LIN {X 0,Y 420.308,Z 548.759,A -85,B 0,C 180,E1 -10290.385,E2 -10290.385} C_VEL
LIN {X 0,Y 420.15,Z 551.033,A -85,B 0,C 180,E1 -10290.92,E2 -10290.92} C_VEL
LIN {X 0,Y 424.128,Z 570.244,A -85,B 0,C 180,E1 -10291.48,E2 -10291.48} C_VEL
LIN {X 0,Y 422.913,Z 658.502,A -85,B 0,C 180,E1 -10293.08,E2 -10293.08} C_VEL
LIN {X 0,Y 422.511,Z 671.225,A -85,B 0,C 180,E1 -10293.497,E2 -10293.497} C_VEL
LIN {X 0,Y 421.973,Z 684.045,A -85,B 0,C 180,E1 -10294.115,E2 -10294.115} C_VEL
LIN {X 0,Y 421.324,Z 696.249,A -85,B 0,C 180,E1 -10294.924,E2 -10294.924} C_VEL
LIN {X 0,Y 420.519,Z 708.11,A -85,B 0,C 180,E1 -10295.936,E2 -10295.936} C_VEL
LIN {X 0,Y 419.769,Z 718.542,A -85,B 0,C 180,E1 -10297.065,E2 -10297.065} C_VEL
LIN {X 0,Y 419.109,Z 728.059,A -85,B 0,C 180,E1 -10298.348,E2 -10298.348} C_VEL
LIN {X 0,Y 418.513,Z 735.947,A -85,B 0,C 180,E1 -10299.651,E2 -10299.651} C_VEL
LIN {X 0,Y 418,Z 742.497,A -85,B 0,C 180,E1 -10300.974,E2 -10300.974} C_VEL
LIN {X 0,Y 417.596,Z 749.006,A -85,B 0,C 180,E1 -10302.629,E2 -10302.629} C_VEL
LIN {X 0,Y 417.299,Z 754.023,A -85,B 0,C 180,E1 -10304.318,E2 -10304.318} C_VEL
LIN {X 0,Y 417.103,Z 757.009,A -85,B 0,C 180,E1 -10305.67,E2 -10305.67} C_VEL
LIN {X 0,Y 416.912,Z 759.823,A -85,B 0,C 180,E1 -10307.603,E2 -10307.603} C_VEL
LIN {X 0,Y 416.814,Z 760.935,A -85,B 0,C 180,E1 -10309.354,E2 -10309.354} C_VEL
LIN {X 0,Y 416.814,Z 760.853,A -85,B 0,C 180,E1 -10310.86,E2 -10310.86} C_VEL
LIN {X 0,Y 416.909,Z 759.474,A -85,B 0,C 180,E1 -10312.639,E2 -10312.639} C_VEL
LIN {X 0,Y 417.117,Z 756.524,A -85,B 0,C 180,E1 -10314.528,E2 -10314.528} C_VEL
LIN {X 0,Y 417.313,Z 752.371,A -85,B 0,C 180,E1 -10316.239,E2 -10316.239} C_VEL
LIN {X 0,Y 417.678,Z 746.51,A -85,B 0,C 180,E1 -10317.994,E2 -10317.994} C_VEL
LIN {X 0,Y 418.041,Z 740.528,A -85,B 0,C 180,E1 -10319.39,E2 -10319.39} C_VEL
LIN {X 0,Y 418.614,Z 732.644,A -85,B 0,C 180,E1 -10320.867,E2 -10320.867} C_VEL
LIN {X 0,Y 419.189,Z 723.962,A -85,B 0,C 180,E1 -10322.175,E2 -10322.175} C_VEL
LIN {X 0,Y 419.91,Z 713.909,A -85,B 0,C 180,E1 -10323.405,E2 -10323.405} C_VEL
LIN {X 0,Y 420.672,Z 703.331,A -85,B 0,C 180,E1 -10324.442,E2 -10324.442} C_VEL
LIN {X 0,Y 421.29,Z 691.58,A -85,B 0,C 180,E1 -10325.353,E2 -10325.353} C_VEL
LIN {X 0,Y 421.916,Z 679.248,A -85,B 0,C 180,E1 -10326.085,E2 -10326.085} C_VEL
LIN {X 0,Y 422.378,Z 666.034,A -85,B 0,C 180,E1 -10326.643,E2 -10326.643} C_VEL
LIN {X 0,Y 422.72,Z 652.404,A -85,B 0,C 180,E1 -10327.003,E2 -10327.003} C_VEL
LIN {X 0,Y 423.711,Z 575.673,A -85,B 0,C 180,E1 -10328.355,E2 -10328.355} C_VEL
LIN {X 0,Y 422.921,Z 571.915,A -85,B 0,C 180,E1 -10328.458,E2 -10328.458} C_VEL
LIN {X 0,Y 420.296,Z 567.48,A -85,B 0,C 180,E1 -10328.654,E2 -10328.654} C_VEL
LIN {X 0,Y 415.703,Z 561.063,A -85,B 0,C 180,E1 -10328.977,E2 -10328.977} C_VEL
LIN {X 0,Y 414.319,Z 557.368,A -85,B 0,C 180,E1 -10329.109,E2 -10329.109} C_VEL
LIN {X 0,Y 412.948,Z 550.435,A -85,B 0,C 180,E1 -10329.328,E2 -10329.328} C_VEL
LIN {X 0,Y 413.198,Z 543.912,A -85,B 0,C 180,E1 -10330.889,E2 -10330.889} C_VEL
LIN {X 0,Y 411.297,Z 533.254,A -85,B 0,C 180,E1 -10333.625,E2 -10333.625} C_VEL
LIN {X 0,Y 411.298,Z 533.253,A -85,B 0,C 180,E1 -10337.167,E2 -10337.167} C_VEL
LIN {X 0,Y 411.289,Z 533.25,A -85,B 0,C 180,E1 -10340.163,E2 -10340.163} C_VEL
LIN {X 0,Y 411.447,Z 533.233,A -85,B 0,C 180,E1 -10343.134,E2 -10343.134} C_VEL
LIN {X 0,Y 411.307,Z 533.251,A -85,B 0,C 180,E1 -10345.1,E2 -10345.1} C_VEL
LIN {X 0,Y 411.511,Z 533.221,A -85,B 0,C 180,E1 -10348.044,E2 -10348.044} C_VEL
LIN {X 0,Y 411.639,Z 533.205,A -85,B 0,C 180,E1 -10350.001,E2 -10350.001} C_VEL
LIN {X 0,Y 411.463,Z 533.235,A -85,B 0,C 180,E1 -10352.939,E2 -10352.939} C_VEL
LIN {X 0,Y 411.449,Z 533.235,A -85,B 0,C 180,E1 -10356.868,E2 -10356.868} C_VEL
LIN {X 0,Y 411.291,Z 533.248,A -85,B 0,C 180,E1 -10359.84,E2 -10359.84} C_VEL
LIN {X 0,Y 411.304,Z 533.254,A -85,B 0,C 180,E1 -10363.106,E2 -10363.106} C_VEL
LIN {X 0,Y 411.262,Z 533.257,A -85,B 0,C 180,E1 -10366.87,E2 -10366.87} C_VEL
LIN {X 0,Y 411.23,Z 533.256,A -85,B 0,C 180,E1 -10369.988,E2 -10369.988} C_VEL
LIN {X 0,Y 411.203,Z 533.267,A -85,B 0,C 180,E1 -10373.149,E2 -10373.149} C_VEL
LIN {X 0,Y 411.238,Z 533.255,A -85,B 0,C 180,E1 -10376.382,E2 -10376.382} C_VEL
LIN {X 0,Y 411.201,Z 533.261,A -85,B 0,C 180,E1 -10379.714,E2 -10379.714} C_VEL
LIN {X 0,Y 411.208,Z 533.265,A -85,B 0,C 180,E1 -10383.157,E2 -10383.157} C_VEL
LIN {X 0,Y 411.194,Z 533.261,A -85,B 0,C 180,E1 -10386.554,E2 -10386.554} C_VEL
LIN {X 0,Y 411.217,Z 533.26,A -85,B 0,C 180,E1 -10389.729,E2 -10389.729} C_VEL
LIN {X 0,Y 411.18,Z 533.267,A -85,B 0,C 180,E1 -10393.134,E2 -10393.134} C_VEL
LIN {X 0,Y 411.171,Z 533.265,A -85,B 0,C 180,E1 -10395.882,E2 -10395.882} C_VEL
LIN {X 0,Y 411.166,Z 533.265,A -85,B 0,C 180,E1 -10398.773,E2 -10398.773} C_VEL
LIN {X 0,Y 411.208,Z 533.262,A -85,B 0,C 180,E1 -10401.833,E2 -10401.833} C_VEL
LIN {X 0,Y 411.215,Z 533.261,A -85,B 0,C 180,E1 -10405.123,E2 -10405.123} C_VEL
LIN {X 0,Y 411.17,Z 533.265,A -85,B 0,C 180,E1 -10408.004,E2 -10408.004} C_VEL
LIN {X 0,Y 411.223,Z 533.263,A -85,B 0,C 180,E1 -10411.411,E2 -10411.411} C_VEL
LIN {X 0,Y 411.242,Z 533.261,A -85,B 0,C 180,E1 -10413.62,E2 -10413.62} C_VEL
LIN {X 0,Y 411.202,Z 533.26,A -85,B 0,C 180,E1 -10416.853,E2 -10416.853} C_VEL
LIN {X 0,Y 411.22,Z 533.26,A -85,B 0,C 180,E1 -10420.051,E2 -10420.051} C_VEL
LIN {X 0,Y 411.269,Z 533.253,A -85,B 0,C 180,E1 -10423.132,E2 -10423.132} C_VEL
LIN {X 0,Y 411.312,Z 533.246,A -85,B 0,C 180,E1 -10426.897,E2 -10426.897} C_VEL
LIN {X 0,Y 411.298,Z 533.25,A -85,B 0,C 180,E1 -10430.162,E2 -10430.162} C_VEL
LIN {X 0,Y 411.459,Z 533.228,A -85,B 0,C 180,E1 -10433.134,E2 -10433.134} C_VEL
LIN {X 0,Y 411.315,Z 533.246,A -85,B 0,C 180,E1 -10435.1,E2 -10435.1} C_VEL
LIN {X 0,Y 411.518,Z 533.225,A -85,B 0,C 180,E1 -10438.043,E2 -10438.043} C_VEL
LIN {X 0,Y 411.647,Z 533.209,A -85,B 0,C 180,E1 -10440.001,E2 -10440.001} C_VEL
LIN {X 0,Y 411.464,Z 533.227,A -85,B 0,C 180,E1 -10442.938,E2 -10442.938} C_VEL
LIN {X 0,Y 411.468,Z 533.226,A -85,B 0,C 180,E1 -10446.867,E2 -10446.867} C_VEL
LIN {X 0,Y 411.362,Z 533.24,A -85,B 0,C 180,E1 -10448.846,E2 -10448.846} C_VEL
LIN {X 0,Y 411.291,Z 533.255,A -85,B 0,C 180,E1 -10451.833,E2 -10451.833} C_VEL
LIN {X 0,Y 411.268,Z 533.251,A -85,B 0,C 180,E1 -10454.853,E2 -10454.853} C_VEL
LIN {X 0,Y 411.258,Z 533.259,A -85,B 0,C 180,E1 -10457.915,E2 -10457.915} C_VEL
LIN {X 0,Y 411.204,Z 533.259,A -85,B 0,C 180,E1 -10461.034,E2 -10461.034} C_VEL
LIN {X 0,Y 411.228,Z 533.262,A -85,B 0,C 180,E1 -10464.216,E2 -10464.216} C_VEL
LIN {X 0,Y 411.267,Z 533.252,A -85,B 0,C 180,E1 -10467.478,E2 -10467.478} C_VEL
LIN {X 0,Y 411.197,Z 533.261,A -85,B 0,C 180,E1 -10470.847,E2 -10470.847} C_VEL
LIN {X 0,Y 411.214,Z 533.263,A -85,B 0,C 180,E1 -10474.333,E2 -10474.333} C_VEL
LIN {X 0,Y 411.198,Z 533.264,A -85,B 0,C 180,E1 -10477.974,E2 -10477.974} C_VEL
LIN {X 0,Y 411.167,Z 533.264,A -85,B 0,C 180,E1 -10481.227,E2 -10481.227} C_VEL
LIN {X 0,Y 411.183,Z 533.267,A -85,B 0,C 180,E1 -10484.49,E2 -10484.49} C_VEL
LIN {X 0,Y 411.185,Z 533.268,A -85,B 0,C 180,E1 -10488.194,E2 -10488.194} C_VEL
LIN {X 0,Y 411.231,Z 533.258,A -85,B 0,C 180,E1 -10490.776,E2 -10490.776} C_VEL
LIN {X 0,Y 411.205,Z 533.266,A -85,B 0,C 180,E1 -10494.471,E2 -10494.471} C_VEL
LIN {X 0,Y 411.215,Z 533.26,A -85,B 0,C 180,E1 -10496.873,E2 -10496.873} C_VEL
LIN {X 0,Y 411.24,Z 533.261,A -85,B 0,C 180,E1 -10500.643,E2 -10500.643} C_VEL
LIN {X 0,Y 411.32,Z 533.412,A -85,B 0,C 180,E1 -10502.353,E2 -10502.353} C_VEL
LIN {X 0,Y 413.758,Z 545.682,A -85,B 0,C 180,E1 -10505.139,E2 -10505.139} C_VEL
LIN {X 0,Y 414.314,Z 549.496,A -85,B 0,C 180,E1 -10505.975,E2 -10505.975} C_VEL
LIN {X 0,Y 413.43,Z 563.343,A -85,B 0,C 180,E1 -10508.823,E2 -10508.823} C_VEL
LIN {X 0,Y 412.789,Z 572.615,A -85,B 0,C 180,E1 -10510.705,E2 -10510.705} C_VEL
LIN {X 0,Y 416.803,Z 598.62,A -85,B 0,C 180,E1 -10511.379,E2 -10511.379} C_VEL
LIN {X 0,Y 415.714,Z 681.281,A -85,B 0,C 180,E1 -10512.885,E2 -10512.885} C_VEL
LIN {X 0,Y 415.188,Z 695.012,A -85,B 0,C 180,E1 -10513.338,E2 -10513.338} C_VEL
LIN {X 0,Y 414.584,Z 707.414,A -85,B 0,C 180,E1 -10513.946,E2 -10513.946} C_VEL
LIN {X 0,Y 413.866,Z 719.311,A -85,B 0,C 180,E1 -10514.738,E2 -10514.738} C_VEL
LIN {X 0,Y 413.089,Z 730.763,A -85,B 0,C 180,E1 -10515.717,E2 -10515.717} C_VEL
LIN {X 0,Y 412.34,Z 741.085,A -85,B 0,C 180,E1 -10516.821,E2 -10516.821} C_VEL
LIN {X 0,Y 411.762,Z 749.532,A -85,B 0,C 180,E1 -10517.93,E2 -10517.93} C_VEL
LIN {X 0,Y 411.046,Z 758.685,A -85,B 0,C 180,E1 -10519.407,E2 -10519.407} C_VEL
LIN {X 0,Y 410.59,Z 766.062,A -85,B 0,C 180,E1 -10520.889,E2 -10520.889} C_VEL
LIN {X 0,Y 410.313,Z 771.055,A -85,B 0,C 180,E1 -10522.123,E2 -10522.123} C_VEL
LIN {X 0,Y 410.101,Z 776.187,A -85,B 0,C 180,E1 -10523.702,E2 -10523.702} C_VEL
LIN {X 0,Y 410.026,Z 779.603,A -85,B 0,C 180,E1 -10525.082,E2 -10525.082} C_VEL
LIN {X 0,Y 409.936,Z 781.513,A -85,B 0,C 180,E1 -10526.066,E2 -10526.066} C_VEL
LIN {X 0,Y 409.929,Z 782.966,A -85,B 0,C 180,E1 -10527.05,E2 -10527.05} C_VEL
LIN {X 0,Y 409.967,Z 783.99,A -85,B 0,C 180,E1 -10528.034,E2 -10528.034} C_VEL
LIN {X 0,Y 409.936,Z 784.617,A -85,B 0,C 180,E1 -10529.016,E2 -10529.016} C_VEL
LIN {X 0,Y 409.926,Z 784.853,A -85,B 0,C 180,E1 -10529.999,E2 -10529.999} C_VEL
LIN {X 0,Y 409.936,Z 784.659,A -85,B 0,C 180,E1 -10530.981,E2 -10530.981} C_VEL
LIN {X 0,Y 409.967,Z 784.052,A -85,B 0,C 180,E1 -10531.963,E2 -10531.963} C_VEL
LIN {X 0,Y 409.935,Z 781.649,A -85,B 0,C 180,E1 -10533.931,E2 -10533.931} C_VEL
LIN {X 0,Y 410.027,Z 778.694,A -85,B 0,C 180,E1 -10535.408,E2 -10535.408} C_VEL
LIN {X 0,Y 410.167,Z 774.695,A -85,B 0,C 180,E1 -10536.887,E2 -10536.887} C_VEL
LIN {X 0,Y 410.483,Z 768.551,A -85,B 0,C 180,E1 -10538.614,E2 -10538.614} C_VEL
LIN {X 0,Y 410.928,Z 761.828,A -85,B 0,C 180,E1 -10540.095,E2 -10540.095} C_VEL
LIN {X 0,Y 411.539,Z 753.491,A -85,B 0,C 180,E1 -10541.574,E2 -10541.574} C_VEL
LIN {X 0,Y 412.26,Z 744.96,A -85,B 0,C 180,E1 -10542.802,E2 -10542.802} C_VEL
LIN {X 0,Y 412.918,Z 735.415,A -85,B 0,C 180,E1 -10543.93,E2 -10543.93} C_VEL
LIN {X 0,Y 413.74,Z 724.036,A -85,B 0,C 180,E1 -10545.012,E2 -10545.012} C_VEL
LIN {X 0,Y 414.488,Z 712.66,A -85,B 0,C 180,E1 -10545.866,E2 -10545.866} C_VEL
LIN {X 0,Y 415.207,Z 701.02,A -85,B 0,C 180,E1 -10546.532,E2 -10546.532} C_VEL
LIN {X 0,Y 415.806,Z 687.714,A -85,B 0,C 180,E1 -10547.076,E2 -10547.076} C_VEL
LIN {X 0,Y 416.248,Z 674.841,A -85,B 0,C 180,E1 -10547.406,E2 -10547.406} C_VEL
LIN {X 0,Y 417.165,Z 597.702,A -85,B 0,C 180,E1 -10548.81,E2 -10548.81} C_VEL
LIN {X 0,Y 412.926,Z 571.903,A -85,B 0,C 180,E1 -10549.543,E2 -10549.543} C_VEL
LIN {X 0,Y 414.272,Z 553.611,A -85,B 0,C 180,E1 -10553.318,E2 -10553.318} C_VEL
LIN {X 0,Y 414.415,Z 549.063,A -85,B 0,C 180,E1 -10554.282,E2 -10554.282} C_VEL
LIN {X 0,Y 412.28,Z 537.945,A -85,B 0,C 180,E1 -10556.853,E2 -10556.853} C_VEL
LIN {X 0,Y 411.275,Z 533.26,A -85,B 0,C 180,E1 -10558.028,E2 -10558.028} C_VEL
LIN {X 0,Y 411.18,Z 533.271,A -85,B 0,C 180,E1 -10561.282,E2 -10561.282} C_VEL
LIN {X 0,Y 411.202,Z 533.262,A -85,B 0,C 180,E1 -10564.332,E2 -10564.332} C_VEL
LIN {X 0,Y 411.2,Z 533.266,A -85,B 0,C 180,E1 -10567.971,E2 -10567.971} C_VEL
LIN {X 0,Y 411.196,Z 533.27,A -85,B 0,C 180,E1 -10571.233,E2 -10571.233} C_VEL
LIN {X 0,Y 411.173,Z 533.268,A -85,B 0,C 180,E1 -10574.488,E2 -10574.488} C_VEL
LIN {X 0,Y 411.192,Z 533.264,A -85,B 0,C 180,E1 -10578.196,E2 -10578.196} C_VEL
LIN {X 0,Y 411.224,Z 533.258,A -85,B 0,C 180,E1 -10580.776,E2 -10580.776} C_VEL
LIN {X 0,Y 411.192,Z 533.263,A -85,B 0,C 180,E1 -10584.47,E2 -10584.47} C_VEL
LIN {X 0,Y 411.199,Z 533.261,A -85,B 0,C 180,E1 -10586.872,E2 -10586.872} C_VEL
LIN {X 0,Y 411.232,Z 533.257,A -85,B 0,C 180,E1 -10590.641,E2 -10590.641} C_VEL
LIN {X 0,Y 411.229,Z 533.26,A -85,B 0,C 180,E1 -10593.618,E2 -10593.618} C_VEL
LIN {X 0,Y 411.193,Z 533.258,A -85,B 0,C 180,E1 -10596.851,E2 -10596.851} C_VEL
LIN {X 0,Y 411.204,Z 533.255,A -85,B 0,C 180,E1 -10600.049,E2 -10600.049} C_VEL
LIN {X 0,Y 411.252,Z 533.259,A -85,B 0,C 180,E1 -10603.13,E2 -10603.13} C_VEL
LIN {X 0,Y 411.302,Z 533.25,A -85,B 0,C 180,E1 -10606.89,E2 -10606.89} C_VEL
LIN {X 0,Y 411.298,Z 533.25,A -85,B 0,C 180,E1 -10610.161,E2 -10610.161} C_VEL
LIN {X 0,Y 411.449,Z 533.231,A -85,B 0,C 180,E1 -10613.132,E2 -10613.132} C_VEL
LIN {X 0,Y 411.303,Z 533.25,A -85,B 0,C 180,E1 -10615.098,E2 -10615.098} C_VEL
LIN {X 0,Y 411.503,Z 533.222,A -85,B 0,C 180,E1 -10618.042,E2 -10618.042} C_VEL
LIN {X 0,Y 411.632,Z 533.209,A -85,B 0,C 180,E1 -10619.999,E2 -10619.999} C_VEL
LIN {X 0,Y 411.457,Z 533.23,A -85,B 0,C 180,E1 -10622.937,E2 -10622.937} C_VEL
LIN {X 0,Y 411.446,Z 533.232,A -85,B 0,C 180,E1 -10626.641,E2 -10626.641} C_VEL
LIN {X 0,Y 411.345,Z 533.246,A -85,B 0,C 180,E1 -10628.845,E2 -10628.845} C_VEL
LIN {X 0,Y 411.29,Z 533.253,A -85,B 0,C 180,E1 -10631.832,E2 -10631.832} C_VEL
LIN {X 0,Y 411.251,Z 533.26,A -85,B 0,C 180,E1 -10634.852,E2 -10634.852} C_VEL
LIN {X 0,Y 411.24,Z 533.261,A -85,B 0,C 180,E1 -10637.915,E2 -10637.915} C_VEL
LIN {X 0,Y 411.184,Z 533.267,A -85,B 0,C 180,E1 -10641.034,E2 -10641.034} C_VEL
LIN {X 0,Y 411.214,Z 533.264,A -85,B 0,C 180,E1 -10644.216,E2 -10644.216} C_VEL
LIN {X 0,Y 411.226,Z 533.274,A -85,B 0,C 180,E1 -10645.904,E2 -10645.904} C_VEL
LIN {X 0,Y 413.319,Z 543.755,A -85,B 0,C 180,E1 -10648.708,E2 -10648.708} C_VEL
LIN {X 0,Y 413.592,Z 546.955,A -85,B 0,C 180,E1 -10649.523,E2 -10649.523} C_VEL
LIN {X 0,Y 413.292,Z 551.196,A -85,B 0,C 180,E1 -10650.554,E2 -10650.554} C_VEL
LIN {X 0,Y 417.493,Z 571.493,A -85,B 0,C 180,E1 -10651.173,E2 -10651.173} C_VEL
LIN {X 0,Y 416.161,Z 658.77,A -85,B 0,C 180,E1 -10652.783,E2 -10652.783} C_VEL
LIN {X 0,Y 415.747,Z 672.146,A -85,B 0,C 180,E1 -10653.234,E2 -10653.234} C_VEL
LIN {X 0,Y 415.188,Z 684.429,A -85,B 0,C 180,E1 -10653.843,E2 -10653.843} C_VEL
LIN {X 0,Y 414.529,Z 695.874,A -85,B 0,C 180,E1 -10654.608,E2 -10654.608} C_VEL
LIN {X 0,Y 413.728,Z 707.768,A -85,B 0,C 180,E1 -10655.632,E2 -10655.632} C_VEL
LIN {X 0,Y 412.988,Z 717.71,A -85,B 0,C 180,E1 -10656.704,E2 -10656.704} C_VEL
LIN {X 0,Y 412.323,Z 726.381,A -85,B 0,C 180,E1 -10657.851,E2 -10657.851} C_VEL
LIN {X 0,Y 411.617,Z 734.604,A -85,B 0,C 180,E1 -10659.178,E2 -10659.178} C_VEL
LIN {X 0,Y 411.099,Z 741.377,A -85,B 0,C 180,E1 -10660.513,E2 -10660.513} C_VEL
LIN {X 0,Y 410.576,Z 748.354,A -85,B 0,C 180,E1 -10662.238,E2 -10662.238} C_VEL
LIN {X 0,Y 410.252,Z 753.685,A -85,B 0,C 180,E1 -10663.989,E2 -10663.989} C_VEL
LIN {X 0,Y 410.068,Z 756.816,A -85,B 0,C 180,E1 -10665.36,E2 -10665.36} C_VEL
LIN {X 0,Y 409.897,Z 759.025,A -85,B 0,C 180,E1 -10666.701,E2 -10666.701} C_VEL
LIN {X 0,Y 409.78,Z 760.437,A -85,B 0,C 180,E1 -10668.022,E2 -10668.022} C_VEL
LIN {X 0,Y 409.737,Z 761.141,A -85,B 0,C 180,E1 -10669.325,E2 -10669.325} C_VEL
LIN {X 0,Y 409.715,Z 761.13,A -85,B 0,C 180,E1 -10670.606,E2 -10670.606} C_VEL
LIN {X 0,Y 409.772,Z 760.268,A -85,B 0,C 180,E1 -10672.086,E2 -10672.086} C_VEL
LIN {X 0,Y 409.918,Z 758.307,A -85,B 0,C 180,E1 -10673.687,E2 -10673.687} C_VEL
LIN {X 0,Y 410.164,Z 754.559,A -85,B 0,C 180,E1 -10675.569,E2 -10675.569} C_VEL
LIN {X 0,Y 410.385,Z 750.416,A -85,B 0,C 180,E1 -10677.049,E2 -10677.049} C_VEL
LIN {X 0,Y 410.775,Z 743.936,A -85,B 0,C 180,E1 -10678.809,E2 -10678.809} C_VEL
LIN {X 0,Y 411.327,Z 736.928,A -85,B 0,C 180,E1 -10680.299,E2 -10680.299} C_VEL
LIN {X 0,Y 411.912,Z 728.57,A -85,B 0,C 180,E1 -10681.721,E2 -10681.721} C_VEL
LIN {X 0,Y 412.61,Z 719.037,A -85,B 0,C 180,E1 -10683.033,E2 -10683.033} C_VEL
LIN {X 0,Y 413.402,Z 708.404,A -85,B 0,C 180,E1 -10684.211,E2 -10684.211} C_VEL
LIN {X 0,Y 414.084,Z 697.588,A -85,B 0,C 180,E1 -10685.163,E2 -10685.163} C_VEL
LIN {X 0,Y 414.765,Z 685.365,A -85,B 0,C 180,E1 -10686.006,E2 -10686.006} C_VEL
LIN {X 0,Y 415.318,Z 673.151,A -85,B 0,C 180,E1 -10686.635,E2 -10686.635} C_VEL
LIN {X 0,Y 415.72,Z 660.345,A -85,B 0,C 180,E1 -10687.087,E2 -10687.087} C_VEL
LIN {X 0,Y 416.051,Z 641.591,A -85,B 0,C 180,E1 -10687.467,E2 -10687.467} C_VEL
LIN {X 0,Y 417.013,Z 571.402,A -85,B 0,C 180,E1 -10688.725,E2 -10688.725} C_VEL
LIN {X 0,Y 414.319,Z 557.368,A -85,B 0,C 180,E1 -10689.109,E2 -10689.109} C_VEL
LIN {X 0,Y 413.378,Z 553.984,A -85,B 0,C 180,E1 -10689.291,E2 -10689.291} C_VEL
LIN {X 0,Y 411.771,Z 550.505,A -85,B 0,C 180,E1 -10689.683,E2 -10689.683} C_VEL
LIN {X 0,Y 409.329,Z 546.791,A -85,B 0,C 180,E1 -10690.406,E2 -10690.406} C_VEL
LIN {X 0,Y 406.714,Z 543.217,A -85,B 0,C 180,E1 -10691.425,E2 -10691.425} C_VEL
LIN {X 0,Y 405.205,Z 539.303,A -85,B 0,C 180,E1 -10692.486,E2 -10692.486} C_VEL
LIN {X 0,Y 404.255,Z 534.131,A -85,B 0,C 180,E1 -10693.851,E2 -10693.851} C_VEL
LIN {X 0,Y 404.277,Z 534.129,A -85,B 0,C 180,E1 -10696.94,E2 -10696.94} C_VEL
LIN {X 0,Y 404.254,Z 534.125,A -85,B 0,C 180,E1 -10699.99,E2 -10699.99} C_VEL
LIN {X 0,Y 404.395,Z 534.113,A -85,B 0,C 180,E1 -10703.014,E2 -10703.014} C_VEL
LIN {X 0,Y 404.279,Z 534.128,A -85,B 0,C 180,E1 -10705.015,E2 -10705.015} C_VEL
LIN {X 0,Y 404.48,Z 534.097,A -85,B 0,C 180,E1 -10708.01,E2 -10708.01} C_VEL
LIN {X 0,Y 404.609,Z 534.081,A -85,B 0,C 180,E1 -10710.001,E2 -10710.001} C_VEL
LIN {X 0,Y 404.42,Z 534.111,A -85,B 0,C 180,E1 -10712.99,E2 -10712.99} C_VEL
LIN {X 0,Y 404.397,Z 534.115,A -85,B 0,C 180,E1 -10716.989,E2 -10716.989} C_VEL
LIN {X 0,Y 404.257,Z 534.125,A -85,B 0,C 180,E1 -10720.013,E2 -10720.013} C_VEL
LIN {X 0,Y 404.265,Z 534.129,A -85,B 0,C 180,E1 -10723.213,E2 -10723.213} C_VEL
LIN {X 0,Y 404.215,Z 534.136,A -85,B 0,C 180,E1 -10727.008,E2 -10727.008} C_VEL
LIN {X 0,Y 404.163,Z 534.137,A -85,B 0,C 180,E1 -10730.353,E2 -10730.353} C_VEL
LIN {X 0,Y 404.169,Z 534.138,A -85,B 0,C 180,E1 -10733.576,E2 -10733.576} C_VEL
LIN {X 0,Y 404.184,Z 534.135,A -85,B 0,C 180,E1 -10735.768,E2 -10735.768} C_VEL
LIN {X 0,Y 404.196,Z 534.132,A -85,B 0,C 180,E1 -10738.001,E2 -10738.001} C_VEL
LIN {X 0,Y 404.141,Z 534.143,A -85,B 0,C 180,E1 -10741.559,E2 -10741.559} C_VEL
LIN {X 0,Y 404.186,Z 534.138,A -85,B 0,C 180,E1 -10745.017,E2 -10745.017} C_VEL
LIN {X 0,Y 404.158,Z 534.138,A -85,B 0,C 180,E1 -10748.758,E2 -10748.758} C_VEL
LIN {X 0,Y 404.127,Z 534.145,A -85,B 0,C 180,E1 -10751.601,E2 -10751.601} C_VEL
LIN {X 0,Y 404.151,Z 534.138,A -85,B 0,C 180,E1 -10754.524,E2 -10754.524} C_VEL
LIN {X 0,Y 404.139,Z 534.146,A -85,B 0,C 180,E1 -10757.297,E2 -10757.297} C_VEL
LIN {X 0,Y 404.172,Z 534.137,A -85,B 0,C 180,E1 -10759.957,E2 -10759.957} C_VEL
LIN {X 0,Y 404.14,Z 534.143,A -85,B 0,C 180,E1 -10763.126,E2 -10763.126} C_VEL
LIN {X 0,Y 404.149,Z 534.139,A -85,B 0,C 180,E1 -10766.189,E2 -10766.189} C_VEL
LIN {X 0,Y 404.15,Z 534.143,A -85,B 0,C 180,E1 -10769.716,E2 -10769.716} C_VEL
LIN {X 0,Y 404.2,Z 534.134,A -85,B 0,C 180,E1 -10773.124,E2 -10773.124} C_VEL
LIN {X 0,Y 404.18,Z 534.139,A -85,B 0,C 180,E1 -10775.335,E2 -10775.335} C_VEL
LIN {X 0,Y 404.144,Z 534.139,A -85,B 0,C 180,E1 -10778.582,E2 -10778.582} C_VEL
LIN {X 0,Y 404.21,Z 534.136,A -85,B 0,C 180,E1 -10781.763,E2 -10781.763} C_VEL
LIN {X 0,Y 404.212,Z 534.13,A -85,B 0,C 180,E1 -10784.883,E2 -10784.883} C_VEL
LIN {X 0,Y 404.262,Z 534.128,A -85,B 0,C 180,E1 -10787.959,E2 -10787.959} C_VEL
LIN {X 0,Y 404.412,Z 534.108,A -85,B 0,C 180,E1 -10792.13,E2 -10792.13} C_VEL
LIN {X 0,Y 404.427,Z 534.108,A -85,B 0,C 180,E1 -10794.016,E2 -10794.016} C_VEL
LIN {X 0,Y 404.487,Z 534.101,A -85,B 0,C 180,E1 -10798.009,E2 -10798.009} C_VEL
LIN {X 0,Y 404.617,Z 534.085,A -85,B 0,C 180,E1 -10800.001,E2 -10800.001} C_VEL
LIN {X 0,Y 404.423,Z 534.104,A -85,B 0,C 180,E1 -10802.989,E2 -10802.989} C_VEL
LIN {X 0,Y 404.42,Z 534.104,A -85,B 0,C 180,E1 -10806.988,E2 -10806.988} C_VEL
LIN {X 0,Y 404.265,Z 534.13,A -85,B 0,C 180,E1 -10810.012,E2 -10810.012} C_VEL
LIN {X 0,Y 404.275,Z 534.123,A -85,B 0,C 180,E1 -10813.212,E2 -10813.212} C_VEL
LIN {X 0,Y 404.224,Z 534.129,A -85,B 0,C 180,E1 -10817.007,E2 -10817.007} C_VEL
LIN {X 0,Y 404.172,Z 534.139,A -85,B 0,C 180,E1 -10820.352,E2 -10820.352} C_VEL
LIN {X 0,Y 404.171,Z 534.137,A -85,B 0,C 180,E1 -10823.575,E2 -10823.575} C_VEL
LIN {X 0,Y 404.191,Z 534.136,A -85,B 0,C 180,E1 -10825.766,E2 -10825.766} C_VEL
LIN {X 0,Y 404.203,Z 534.137,A -85,B 0,C 180,E1 -10828,E2 -10828} C_VEL
LIN {X 0,Y 404.147,Z 534.14,A -85,B 0,C 180,E1 -10831.558,E2 -10831.558} C_VEL
LIN {X 0,Y 404.193,Z 534.133,A -85,B 0,C 180,E1 -10835.016,E2 -10835.016} C_VEL
LIN {X 0,Y 404.156,Z 534.139,A -85,B 0,C 180,E1 -10838.757,E2 -10838.757} C_VEL
LIN {X 0,Y 404.126,Z 534.142,A -85,B 0,C 180,E1 -10841.599,E2 -10841.599} C_VEL
LIN {X 0,Y 404.152,Z 534.142,A -85,B 0,C 180,E1 -10844.521,E2 -10844.521} C_VEL
LIN {X 0,Y 404.144,Z 534.139,A -85,B 0,C 180,E1 -10847.295,E2 -10847.295} C_VEL
LIN {X 0,Y 404.177,Z 534.138,A -85,B 0,C 180,E1 -10849.955,E2 -10849.955} C_VEL
LIN {X 0,Y 404.146,Z 534.139,A -85,B 0,C 180,E1 -10853.124,E2 -10853.124} C_VEL
LIN {X 0,Y 404.152,Z 534.143,A -85,B 0,C 180,E1 -10856.187,E2 -10856.187} C_VEL
LIN {X 0,Y 404.153,Z 534.142,A -85,B 0,C 180,E1 -10859.714,E2 -10859.714} C_VEL
LIN {X 0,Y 404.264,Z 534.188,A -85,B 0,C 180,E1 -10862.069,E2 -10862.069} C_VEL
LIN {X 0,Y 406.758,Z 546.654,A -85,B 0,C 180,E1 -10864.955,E2 -10864.955} C_VEL
LIN {X 0,Y 407.331,Z 551.967,A -85,B 0,C 180,E1 -10866.129,E2 -10866.129} C_VEL
LIN {X 0,Y 406.236,Z 566.241,A -85,B 0,C 180,E1 -10869.103,E2 -10869.103} C_VEL
LIN {X 0,Y 405.851,Z 572.477,A -85,B 0,C 180,E1 -10870.393,E2 -10870.393} C_VEL
LIN {X 0,Y 410.04,Z 599.227,A -85,B 0,C 180,E1 -10871.094,E2 -10871.094} C_VEL
LIN {X 0,Y 408.937,Z 680.326,A -85,B 0,C 180,E1 -10872.592,E2 -10872.592} C_VEL
LIN {X 0,Y 408.397,Z 693.542,A -85,B 0,C 180,E1 -10873.02,E2 -10873.02} C_VEL
LIN {X 0,Y 407.823,Z 705.724,A -85,B 0,C 180,E1 -10873.608,E2 -10873.608} C_VEL
LIN {X 0,Y 407.099,Z 717.225,A -85,B 0,C 180,E1 -10874.35,E2 -10874.35} C_VEL
LIN {X 0,Y 406.253,Z 729.041,A -85,B 0,C 180,E1 -10875.344,E2 -10875.344} C_VEL
LIN {X 0,Y 405.518,Z 739.642,A -85,B 0,C 180,E1 -10876.468,E2 -10876.468} C_VEL
LIN {X 0,Y 404.79,Z 749.191,A -85,B 0,C 180,E1 -10877.719,E2 -10877.719} C_VEL
LIN {X 0,Y 404.026,Z 758.373,A -85,B 0,C 180,E1 -10879.221,E2 -10879.221} C_VEL
LIN {X 0,Y 403.534,Z 765.771,A -85,B 0,C 180,E1 -10880.728,E2 -10880.728} C_VEL
LIN {X 0,Y 403.248,Z 770.783,A -85,B 0,C 180,E1 -10881.984,E2 -10881.984} C_VEL
LIN {X 0,Y 402.991,Z 776.397,A -85,B 0,C 180,E1 -10883.754,E2 -10883.754} C_VEL
LIN {X 0,Y 402.939,Z 779.362,A -85,B 0,C 180,E1 -10884.996,E2 -10884.996} C_VEL
LIN {X 0,Y 402.857,Z 781.279,A -85,B 0,C 180,E1 -10885.997,E2 -10885.997} C_VEL
LIN {X 0,Y 402.828,Z 782.743,A -85,B 0,C 180,E1 -10886.998,E2 -10886.998} C_VEL
LIN {X 0,Y 402.866,Z 783.772,A -85,B 0,C 180,E1 -10887.999,E2 -10887.999} C_VEL
LIN {X 0,Y 402.863,Z 784.405,A -85,B 0,C 180,E1 -10888.999,E2 -10888.999} C_VEL
LIN {X 0,Y 402.851,Z 784.646,A -85,B 0,C 180,E1 -10889.999,E2 -10889.999} C_VEL
LIN {X 0,Y 402.863,Z 784.46,A -85,B 0,C 180,E1 -10890.998,E2 -10890.998} C_VEL
LIN {X 0,Y 402.865,Z 783.857,A -85,B 0,C 180,E1 -10891.998,E2 -10891.998} C_VEL
LIN {X 0,Y 402.856,Z 781.46,A -85,B 0,C 180,E1 -10894,E2 -10894} C_VEL
LIN {X 0,Y 402.928,Z 778.51,A -85,B 0,C 180,E1 -10895.504,E2 -10895.504} C_VEL
LIN {X 0,Y 403.081,Z 774.517,A -85,B 0,C 180,E1 -10897.009,E2 -10897.009} C_VEL
LIN {X 0,Y 403.424,Z 768.389,A -85,B 0,C 180,E1 -10898.766,E2 -10898.766} C_VEL
LIN {X 0,Y 403.916,Z 761.684,A -85,B 0,C 180,E1 -10900.272,E2 -10900.272} C_VEL
LIN {X 0,Y 404.567,Z 753.369,A -85,B 0,C 180,E1 -10901.776,E2 -10901.776} C_VEL
LIN {X 0,Y 405.311,Z 744.864,A -85,B 0,C 180,E1 -10903.026,E2 -10903.026} C_VEL
LIN {X 0,Y 406.019,Z 734.862,A -85,B 0,C 180,E1 -10904.225,E2 -10904.225} C_VEL
LIN {X 0,Y 406.875,Z 723.995,A -85,B 0,C 180,E1 -10905.271,E2 -10905.271} C_VEL
LIN {X 0,Y 407.653,Z 712.659,A -85,B 0,C 180,E1 -10906.139,E2 -10906.139} C_VEL
LIN {X 0,Y 408.422,Z 701.118,A -85,B 0,C 180,E1 -10906.815,E2 -10906.815} C_VEL
LIN {X 0,Y 409.017,Z 688.849,A -85,B 0,C 180,E1 -10907.337,E2 -10907.337} C_VEL
LIN {X 0,Y 409.51,Z 675.371,A -85,B 0,C 180,E1 -10907.702,E2 -10907.702} C_VEL
LIN {X 0,Y 410.455,Z 598.516,A -85,B 0,C 180,E1 -10909.13,E2 -10909.13} C_VEL
LIN {X 0,Y 406.531,Z 574.741,A -85,B 0,C 180,E1 -10909.806,E2 -10909.806} C_VEL
LIN {X 0,Y 406.056,Z 571.753,A -85,B 0,C 180,E1 -10909.9,E2 -10909.9} C_VEL
LIN {X 0,Y 407.316,Z 555.213,A -85,B 0,C 180,E1 -10913.38,E2 -10913.38} C_VEL
LIN {X 0,Y 407.612,Z 551.828,A -85,B 0,C 180,E1 -10914.1,E2 -10914.1} C_VEL
LIN {X 0,Y 406.045,Z 542.586,A -85,B 0,C 180,E1 -10916.251,E2 -10916.251} C_VEL
LIN {X 0,Y 404.206,Z 534.141,A -85,B 0,C 180,E1 -10918.35,E2 -10918.35} C_VEL
LIN {X 0,Y 404.136,Z 534.15,A -85,B 0,C 180,E1 -10921.556,E2 -10921.556} C_VEL
LIN {X 0,Y 404.182,Z 534.139,A -85,B 0,C 180,E1 -10925.014,E2 -10925.014} C_VEL
LIN {X 0,Y 404.159,Z 534.143,A -85,B 0,C 180,E1 -10928.754,E2 -10928.754} C_VEL
LIN {X 0,Y 404.146,Z 534.149,A -85,B 0,C 180,E1 -10931.603,E2 -10931.603} C_VEL
LIN {X 0,Y 404.143,Z 534.144,A -85,B 0,C 180,E1 -10934.521,E2 -10934.521} C_VEL
LIN {X 0,Y 404.164,Z 534.141,A -85,B 0,C 180,E1 -10937.299,E2 -10937.299} C_VEL
LIN {X 0,Y 404.162,Z 534.139,A -85,B 0,C 180,E1 -10939.954,E2 -10939.954} C_VEL
LIN {X 0,Y 404.133,Z 534.141,A -85,B 0,C 180,E1 -10943.123,E2 -10943.123} C_VEL
LIN {X 0,Y 404.137,Z 534.14,A -85,B 0,C 180,E1 -10946.186,E2 -10946.186} C_VEL
LIN {X 0,Y 404.145,Z 534.142,A -85,B 0,C 180,E1 -10949.714,E2 -10949.714} C_VEL
LIN {X 0,Y 404.186,Z 534.133,A -85,B 0,C 180,E1 -10953.122,E2 -10953.122} C_VEL
LIN {X 0,Y 404.168,Z 534.141,A -85,B 0,C 180,E1 -10955.333,E2 -10955.333} C_VEL
LIN {X 0,Y 404.129,Z 534.143,A -85,B 0,C 180,E1 -10958.58,E2 -10958.58} C_VEL
LIN {X 0,Y 404.2,Z 534.137,A -85,B 0,C 180,E1 -10961.761,E2 -10961.761} C_VEL
LIN {X 0,Y 404.197,Z 534.13,A -85,B 0,C 180,E1 -10964.881,E2 -10964.881} C_VEL
LIN {X 0,Y 404.259,Z 534.122,A -85,B 0,C 180,E1 -10967.958,E2 -10967.958} C_VEL
LIN {X 0,Y 404.422,Z 534.104,A -85,B 0,C 180,E1 -10972.099,E2 -10972.099} C_VEL
LIN {X 0,Y 404.413,Z 534.107,A -85,B 0,C 180,E1 -10974.014,E2 -10974.014} C_VEL
LIN {X 0,Y 404.472,Z 534.098,A -85,B 0,C 180,E1 -10978.008,E2 -10978.008} C_VEL
LIN {X 0,Y 404.602,Z 534.085,A -85,B 0,C 180,E1 -10979.999,E2 -10979.999} C_VEL
LIN {X 0,Y 404.414,Z 534.108,A -85,B 0,C 180,E1 -10982.988,E2 -10982.988} C_VEL
LIN {X 0,Y 404.396,Z 534.11,A -85,B 0,C 180,E1 -10986.64,E2 -10986.64} C_VEL
LIN {X 0,Y 404.284,Z 534.126,A -85,B 0,C 180,E1 -10989.001,E2 -10989.001} C_VEL
LIN {X 0,Y 404.26,Z 534.129,A -85,B 0,C 180,E1 -10992.041,E2 -10992.041} C_VEL
LIN {X 0,Y 404.196,Z 534.141,A -85,B 0,C 180,E1 -10995.118,E2 -10995.118} C_VEL
LIN {X 0,Y 404.198,Z 534.137,A -85,B 0,C 180,E1 -10998.238,E2 -10998.238} C_VEL
LIN {X 0,Y 404.126,Z 534.144,A -85,B 0,C 180,E1 -11001.419,E2 -11001.419} C_VEL
LIN {X 0,Y 404.162,Z 534.142,A -85,B 0,C 180,E1 -11004.666,E2 -11004.666} C_VEL
LIN {X 0,Y 404.213,Z 534.268,A -85,B 0,C 180,E1 -11005.618,E2 -11005.618} C_VEL
LIN {X 0,Y 406.452,Z 545.449,A -85,B 0,C 180,E1 -11008.673,E2 -11008.673} C_VEL
LIN {X 0,Y 406.647,Z 548.694,A -85,B 0,C 180,E1 -11009.508,E2 -11009.508} C_VEL
LIN {X 0,Y 406.42,Z 551.465,A -85,B 0,C 180,E1 -11010.191,E2 -11010.191} C_VEL
LIN {X 0,Y 410.796,Z 572.376,A -85,B 0,C 180,E1 -11010.844,E2 -11010.844} C_VEL
LIN {X 0,Y 409.46,Z 658.298,A -85,B 0,C 180,E1 -11012.455,E2 -11012.455} C_VEL
LIN {X 0,Y 409.008,Z 671.555,A -85,B 0,C 180,E1 -11012.899,E2 -11012.899} C_VEL
LIN {X 0,Y 408.427,Z 684.503,A -85,B 0,C 180,E1 -11013.543,E2 -11013.543} C_VEL
LIN {X 0,Y 407.757,Z 695.653,A -85,B 0,C 180,E1 -11014.294,E2 -11014.294} C_VEL
LIN {X 0,Y 406.884,Z 707.839,A -85,B 0,C 180,E1 -11015.354,E2 -11015.354} C_VEL
LIN {X 0,Y 406.056,Z 718.349,A -85,B 0,C 180,E1 -11016.509,E2 -11016.509} C_VEL
LIN {X 0,Y 405.281,Z 727.874,A -85,B 0,C 180,E1 -11017.82,E2 -11017.82} C_VEL
LIN {X 0,Y 404.496,Z 736.896,A -85,B 0,C 180,E1 -11019.358,E2 -11019.358} C_VEL
LIN {X 0,Y 403.956,Z 743.334,A -85,B 0,C 180,E1 -11020.723,E2 -11020.723} C_VEL
LIN {X 0,Y 403.502,Z 749.804,A -85,B 0,C 180,E1 -11022.46,E2 -11022.46} C_VEL
LIN {X 0,Y 403.143,Z 754.741,A -85,B 0,C 180,E1 -11024.212,E2 -11024.212} C_VEL
LIN {X 0,Y 402.932,Z 757.907,A -85,B 0,C 180,E1 -11025.761,E2 -11025.761} C_VEL
LIN {X 0,Y 402.764,Z 759.834,A -85,B 0,C 180,E1 -11027.127,E2 -11027.127} C_VEL
LIN {X 0,Y 402.648,Z 761.08,A -85,B 0,C 180,E1 -11028.636,E2 -11028.636} C_VEL
LIN {X 0,Y 402.636,Z 761.409,A -85,B 0,C 180,E1 -11030.175,E2 -11030.175} C_VEL
LIN {X 0,Y 402.663,Z 760.756,A -85,B 0,C 180,E1 -11031.759,E2 -11031.759} C_VEL
LIN {X 0,Y 402.83,Z 758.68,A -85,B 0,C 180,E1 -11033.619,E2 -11033.619} C_VEL
LIN {X 0,Y 403.094,Z 754.948,A -85,B 0,C 180,E1 -11035.573,E2 -11035.573} C_VEL
LIN {X 0,Y 403.345,Z 750.116,A -85,B 0,C 180,E1 -11037.308,E2 -11037.308} C_VEL
LIN {X 0,Y 403.706,Z 744.546,A -85,B 0,C 180,E1 -11038.842,E2 -11038.842} C_VEL
LIN {X 0,Y 404.281,Z 737.598,A -85,B 0,C 180,E1 -11040.364,E2 -11040.364} C_VEL
LIN {X 0,Y 404.856,Z 729.647,A -85,B 0,C 180,E1 -11041.77,E2 -11041.77} C_VEL
LIN {X 0,Y 405.558,Z 720.451,A -85,B 0,C 180,E1 -11043.083,E2 -11043.083} C_VEL
LIN {X 0,Y 406.275,Z 710.819,A -85,B 0,C 180,E1 -11044.205,E2 -11044.205} C_VEL
LIN {X 0,Y 407.084,Z 699.66,A -85,B 0,C 180,E1 -11045.252,E2 -11045.252} C_VEL
LIN {X 0,Y 407.74,Z 687.826,A -85,B 0,C 180,E1 -11046.118,E2 -11046.118} C_VEL
LIN {X 0,Y 408.405,Z 674.997,A -85,B 0,C 180,E1 -11046.82,E2 -11046.82} C_VEL
LIN {X 0,Y 408.897,Z 661.901,A -85,B 0,C 180,E1 -11047.318,E2 -11047.318} C_VEL
LIN {X 0,Y 409.207,Z 645.928,A -85,B 0,C 180,E1 -11047.669,E2 -11047.669} C_VEL
LIN {X 0,Y 410.151,Z 571.641,A -85,B 0,C 180,E1 -11049.029,E2 -11049.029} C_VEL
LIN {X 0,Y 406.012,Z 550.636,A -85,B 0,C 180,E1 -11049.647,E2 -11049.647} C_VEL
LIN {X 0,Y 406.295,Z 545.804,A -85,B 0,C 180,E1 -11050.814,E2 -11050.814} C_VEL
LIN {X 0,Y 405.205,Z 539.303,A -85,B 0,C 180,E1 -11052.486,E2 -11052.486} C_VEL
LIN {X 0,Y 404.213,Z 537.638,A -85,B 0,C 180,E1 -11052.983,E2 -11052.983} C_VEL
LIN {X 0,Y 400.968,Z 535.894,A -85,B 0,C 180,E1 -11053.796,E2 -11053.796} C_VEL
LIN {X 0,Y 397.888,Z 535.128,A -85,B 0,C 180,E1 -11054.658,E2 -11054.658} C_VEL
LIN {X 0,Y 397.165,Z 535.011,A -85,B 0,C 180,E1 -11055.227,E2 -11055.227} C_VEL
LIN {X 0,Y 397.214,Z 535.003,A -85,B 0,C 180,E1 -11057.743,E2 -11057.743} C_VEL
LIN {X 0,Y 397.248,Z 535.005,A -85,B 0,C 180,E1 -11060.84,E2 -11060.84} C_VEL
LIN {X 0,Y 397.366,Z 534.983,A -85,B 0,C 180,E1 -11063.91,E2 -11063.91} C_VEL
LIN {X 0,Y 397.449,Z 534.973,A -85,B 0,C 180,E1 -11067.975,E2 -11067.975} C_VEL
LIN {X 0,Y 397.578,Z 534.957,A -85,B 0,C 180,E1 -11070.001,E2 -11070.001} C_VEL
LIN {X 0,Y 397.378,Z 534.988,A -85,B 0,C 180,E1 -11073.043,E2 -11073.043} C_VEL
LIN {X 0,Y 397.368,Z 534.983,A -85,B 0,C 180,E1 -11076.093,E2 -11076.093} C_VEL
LIN {X 0,Y 397.251,Z 535.003,A -85,B 0,C 180,E1 -11079.163,E2 -11079.163} C_VEL
LIN {X 0,Y 397.218,Z 535.002,A -85,B 0,C 180,E1 -11082.26,E2 -11082.26} C_VEL
LIN {X 0,Y 397.179,Z 535.01,A -85,B 0,C 180,E1 -11085.393,E2 -11085.393} C_VEL
LIN {X 0,Y 397.161,Z 535.01,A -85,B 0,C 180,E1 -11088.575,E2 -11088.575} C_VEL
LIN {X 0,Y 397.097,Z 535.017,A -85,B 0,C 180,E1 -11091.82,E2 -11091.82} C_VEL
LIN {X 0,Y 397.157,Z 535.016,A -85,B 0,C 180,E1 -11095.133,E2 -11095.133} C_VEL
LIN {X 0,Y 397.163,Z 535.01,A -85,B 0,C 180,E1 -11097.777,E2 -11097.777} C_VEL
LIN {X 0,Y 397.08,Z 535.022,A -85,B 0,C 180,E1 -11100.884,E2 -11100.884} C_VEL
LIN {X 0,Y 397.127,Z 535.013,A -85,B 0,C 180,E1 -11104.495,E2 -11104.495} C_VEL
LIN {X 0,Y 397.105,Z 535.016,A -85,B 0,C 180,E1 -11108.276,E2 -11108.276} C_VEL
LIN {X 0,Y 397.092,Z 535.02,A -85,B 0,C 180,E1 -11110.91,E2 -11110.91} C_VEL
LIN {X 0,Y 397.106,Z 535.019,A -85,B 0,C 180,E1 -11113.649,E2 -11113.649} C_VEL
LIN {X 0,Y 397.105,Z 535.016,A -85,B 0,C 180,E1 -11116.522,E2 -11116.522} C_VEL
LIN {X 0,Y 397.117,Z 535.014,A -85,B 0,C 180,E1 -11120.424,E2 -11120.424} C_VEL
LIN {X 0,Y 397.112,Z 535.015,A -85,B 0,C 180,E1 -11124.266,E2 -11124.266} C_VEL
LIN {X 0,Y 397.119,Z 535.014,A -85,B 0,C 180,E1 -11126.728,E2 -11126.728} C_VEL
LIN {X 0,Y 397.129,Z 535.013,A -85,B 0,C 180,E1 -11130.297,E2 -11130.297} C_VEL
LIN {X 0,Y 397.199,Z 535.004,A -85,B 0,C 180,E1 -11132.611,E2 -11132.611} C_VEL
LIN {X 0,Y 397.134,Z 535.015,A -85,B 0,C 180,E1 -11135.982,E2 -11135.982} C_VEL
LIN {X 0,Y 397.15,Z 535.016,A -85,B 0,C 180,E1 -11139.703,E2 -11139.703} C_VEL
LIN {X 0,Y 397.188,Z 535.005,A -85,B 0,C 180,E1 -11142.846,E2 -11142.846} C_VEL
LIN {X 0,Y 397.235,Z 534.999,A -85,B 0,C 180,E1 -11146.704,E2 -11146.704} C_VEL
LIN {X 0,Y 397.223,Z 535.007,A -85,B 0,C 180,E1 -11149.81,E2 -11149.81} C_VEL
LIN {X 0,Y 397.357,Z 534.984,A -85,B 0,C 180,E1 -11152.889,E2 -11152.889} C_VEL
LIN {X 0,Y 397.26,Z 534.996,A -85,B 0,C 180,E1 -11154.926,E2 -11154.926} C_VEL
LIN {X 0,Y 397.456,Z 534.977,A -85,B 0,C 180,E1 -11157.974,E2 -11157.974} C_VEL
LIN {X 0,Y 397.586,Z 534.961,A -85,B 0,C 180,E1 -11160.001,E2 -11160.001} C_VEL
LIN {X 0,Y 397.382,Z 534.981,A -85,B 0,C 180,E1 -11163.042,E2 -11163.042} C_VEL
LIN {X 0,Y 397.372,Z 534.983,A -85,B 0,C 180,E1 -11167.112,E2 -11167.112} C_VEL
LIN {X 0,Y 397.224,Z 535.005,A -85,B 0,C 180,E1 -11170.191,E2 -11170.191} C_VEL
LIN {X 0,Y 397.235,Z 535,A -85,B 0,C 180,E1 -11173.321,E2 -11173.321} C_VEL
LIN {X 0,Y 397.19,Z 535.005,A -85,B 0,C 180,E1 -11177.155,E2 -11177.155} C_VEL
LIN {X 0,Y 397.111,Z 535.016,A -85,B 0,C 180,E1 -11180.73,E2 -11180.73} C_VEL
LIN {X 0,Y 397.136,Z 535.018,A -85,B 0,C 180,E1 -11184.019,E2 -11184.019} C_VEL
LIN {X 0,Y 397.202,Z 535.004,A -85,B 0,C 180,E1 -11187.39,E2 -11187.39} C_VEL
LIN {X 0,Y 397.086,Z 535.018,A -85,B 0,C 180,E1 -11190.882,E2 -11190.882} C_VEL
LIN {X 0,Y 397.134,Z 535.016,A -85,B 0,C 180,E1 -11194.493,E2 -11194.493} C_VEL
LIN {X 0,Y 397.106,Z 535.022,A -85,B 0,C 180,E1 -11198.275,E2 -11198.275} C_VEL
LIN {X 0,Y 397.094,Z 535.018,A -85,B 0,C 180,E1 -11200.909,E2 -11200.909} C_VEL
LIN {X 0,Y 397.107,Z 535.016,A -85,B 0,C 180,E1 -11203.648,E2 -11203.648} C_VEL
LIN {X 0,Y 397.11,Z 535.02,A -85,B 0,C 180,E1 -11206.52,E2 -11206.52} C_VEL
LIN {X 0,Y 397.123,Z 535.02,A -85,B 0,C 180,E1 -11210.422,E2 -11210.422} C_VEL
LIN {X 0,Y 397.116,Z 535.02,A -85,B 0,C 180,E1 -11214.265,E2 -11214.265} C_VEL
LIN {X 0,Y 397.122,Z 535.017,A -85,B 0,C 180,E1 -11216.726,E2 -11216.726} C_VEL
LIN {X 0,Y 397.132,Z 535.017,A -85,B 0,C 180,E1 -11220.295,E2 -11220.295} C_VEL
LIN {X 0,Y 397.209,Z 535.148,A -85,B 0,C 180,E1 -11221.819,E2 -11221.819} C_VEL
LIN {X 0,Y 399.74,Z 547.612,A -85,B 0,C 180,E1 -11224.763,E2 -11224.763} C_VEL
LIN {X 0,Y 400.429,Z 552.522,A -85,B 0,C 180,E1 -11225.877,E2 -11225.877} C_VEL
LIN {X 0,Y 399.318,Z 566.655,A -85,B 0,C 180,E1 -11228.877,E2 -11228.877} C_VEL
LIN {X 0,Y 398.934,Z 572.26,A -85,B 0,C 180,E1 -11230.057,E2 -11230.057} C_VEL
LIN {X 0,Y 403.283,Z 600.121,A -85,B 0,C 180,E1 -11230.81,E2 -11230.81} C_VEL
LIN {X 0,Y 402.122,Z 680.24,A -85,B 0,C 180,E1 -11232.321,E2 -11232.321} C_VEL
LIN {X 0,Y 401.571,Z 693.412,A -85,B 0,C 180,E1 -11232.756,E2 -11232.756} C_VEL
LIN {X 0,Y 400.948,Z 705.008,A -85,B 0,C 180,E1 -11233.319,E2 -11233.319} C_VEL
LIN {X 0,Y 400.239,Z 716.632,A -85,B 0,C 180,E1 -11234.074,E2 -11234.074} C_VEL
LIN {X 0,Y 399.323,Z 728.552,A -85,B 0,C 180,E1 -11235.083,E2 -11235.083} C_VEL
LIN {X 0,Y 398.54,Z 739.68,A -85,B 0,C 180,E1 -11236.283,E2 -11236.283} C_VEL
LIN {X 0,Y 397.833,Z 748.817,A -85,B 0,C 180,E1 -11237.501,E2 -11237.501} C_VEL
LIN {X 0,Y 397.02,Z 758.042,A -85,B 0,C 180,E1 -11239.029,E2 -11239.029} C_VEL
LIN {X 0,Y 396.505,Z 765.469,A -85,B 0,C 180,E1 -11240.562,E2 -11240.562} C_VEL
LIN {X 0,Y 396.2,Z 770.503,A -85,B 0,C 180,E1 -11241.84,E2 -11241.84} C_VEL
LIN {X 0,Y 395.97,Z 775.383,A -85,B 0,C 180,E1 -11243.374,E2 -11243.374} C_VEL
LIN {X 0,Y 395.852,Z 779.118,A -85,B 0,C 180,E1 -11244.906,E2 -11244.906} C_VEL
LIN {X 0,Y 395.779,Z 781.042,A -85,B 0,C 180,E1 -11245.925,E2 -11245.925} C_VEL
LIN {X 0,Y 395.731,Z 782.518,A -85,B 0,C 180,E1 -11246.944,E2 -11246.944} C_VEL
LIN {X 0,Y 395.764,Z 783.553,A -85,B 0,C 180,E1 -11247.963,E2 -11247.963} C_VEL
LIN {X 0,Y 395.792,Z 784.193,A -85,B 0,C 180,E1 -11248.981,E2 -11248.981} C_VEL
LIN {X 0,Y 395.779,Z 784.439,A -85,B 0,C 180,E1 -11249.999,E2 -11249.999} C_VEL
LIN {X 0,Y 395.791,Z 784.263,A -85,B 0,C 180,E1 -11251.016,E2 -11251.016} C_VEL
LIN {X 0,Y 395.763,Z 783.663,A -85,B 0,C 180,E1 -11252.034,E2 -11252.034} C_VEL
LIN {X 0,Y 395.778,Z 781.277,A -85,B 0,C 180,E1 -11254.072,E2 -11254.072} C_VEL
LIN {X 0,Y 395.832,Z 777.869,A -85,B 0,C 180,E1 -11255.811,E2 -11255.811} C_VEL
LIN {X 0,Y 396.08,Z 772.77,A -85,B 0,C 180,E1 -11257.646,E2 -11257.646} C_VEL
LIN {X 0,Y 396.52,Z 766.2,A -85,B 0,C 180,E1 -11259.435,E2 -11259.435} C_VEL
LIN {X 0,Y 397.042,Z 758.993,A -85,B 0,C 180,E1 -11260.968,E2 -11260.968} C_VEL
LIN {X 0,Y 397.892,Z 750.033,A -85,B 0,C 180,E1 -11262.495,E2 -11262.495} C_VEL
LIN {X 0,Y 398.641,Z 741.039,A -85,B 0,C 180,E1 -11263.742,E2 -11263.742} C_VEL
LIN {X 0,Y 399.466,Z 731.08,A -85,B 0,C 180,E1 -11264.869,E2 -11264.869} C_VEL
LIN {X 0,Y 400.382,Z 719.43,A -85,B 0,C 180,E1 -11265.917,E2 -11265.917} C_VEL
LIN {X 0,Y 401.16,Z 708.8,A -85,B 0,C 180,E1 -11266.669,E2 -11266.669} C_VEL
LIN {X 0,Y 401.906,Z 696.055,A -85,B 0,C 180,E1 -11267.358,E2 -11267.358} C_VEL
LIN {X 0,Y 402.507,Z 683.436,A -85,B 0,C 180,E1 -11267.823,E2 -11267.823} C_VEL
LIN {X 0,Y 402.963,Z 664.455,A -85,B 0,C 180,E1 -11268.229,E2 -11268.229} C_VEL
LIN {X 0,Y 403.737,Z 598.983,A -85,B 0,C 180,E1 -11269.477,E2 -11269.477} C_VEL
LIN {X 0,Y 400.217,Z 577.273,A -85,B 0,C 180,E1 -11270.106,E2 -11270.106} C_VEL
LIN {X 0,Y 399.194,Z 571.574,A -85,B 0,C 180,E1 -11270.282,E2 -11270.282} C_VEL
LIN {X 0,Y 400.71,Z 553.282,A -85,B 0,C 180,E1 -11274.213,E2 -11274.213} C_VEL
LIN {X 0,Y 399.144,Z 544.101,A -85,B 0,C 180,E1 -11276.395,E2 -11276.395} C_VEL
LIN {X 0,Y 397.141,Z 535.02,A -85,B 0,C 180,E1 -11278.685,E2 -11278.685} C_VEL
LIN {X 0,Y 397.075,Z 535.025,A -85,B 0,C 180,E1 -11282.07,E2 -11282.07} C_VEL
LIN {X 0,Y 397.116,Z 535.021,A -85,B 0,C 180,E1 -11285.502,E2 -11285.502} C_VEL
LIN {X 0,Y 397.133,Z 535.018,A -85,B 0,C 180,E1 -11288.861,E2 -11288.861} C_VEL
LIN {X 0,Y 397.11,Z 535.02,A -85,B 0,C 180,E1 -11292.259,E2 -11292.259} C_VEL
LIN {X 0,Y 397.083,Z 535.024,A -85,B 0,C 180,E1 -11295.067,E2 -11295.067} C_VEL
LIN {X 0,Y 397.103,Z 535.021,A -85,B 0,C 180,E1 -11298.013,E2 -11298.013} C_VEL
LIN {X 0,Y 397.13,Z 535.017,A -85,B 0,C 180,E1 -11301.136,E2 -11301.136} C_VEL
LIN {X 0,Y 397.112,Z 535.017,A -85,B 0,C 180,E1 -11304.495,E2 -11304.495} C_VEL
LIN {X 0,Y 397.072,Z 535.022,A -85,B 0,C 180,E1 -11307.927,E2 -11307.927} C_VEL
LIN {X 0,Y 397.118,Z 535.019,A -85,B 0,C 180,E1 -11311.456,E2 -11311.456} C_VEL
LIN {X 0,Y 397.143,Z 535.013,A -85,B 0,C 180,E1 -11314.486,E2 -11314.486} C_VEL
LIN {X 0,Y 397.099,Z 535.015,A -85,B 0,C 180,E1 -11317.085,E2 -11317.085} C_VEL
LIN {X 0,Y 397.138,Z 535.006,A -85,B 0,C 180,E1 -11320.352,E2 -11320.352} C_VEL
LIN {X 0,Y 397.156,Z 535.01,A -85,B 0,C 180,E1 -11323.552,E2 -11323.552} C_VEL
LIN {X 0,Y 397.217,Z 535.004,A -85,B 0,C 180,E1 -11326.702,E2 -11326.702} C_VEL
LIN {X 0,Y 397.218,Z 535.006,A -85,B 0,C 180,E1 -11329.808,E2 -11329.808} C_VEL
LIN {X 0,Y 397.353,Z 534.985,A -85,B 0,C 180,E1 -11332.887,E2 -11332.887} C_VEL
LIN {X 0,Y 397.246,Z 535.001,A -85,B 0,C 180,E1 -11334.925,E2 -11334.925} C_VEL
LIN {X 0,Y 397.441,Z 534.974,A -85,B 0,C 180,E1 -11337.973,E2 -11337.973} C_VEL
LIN {X 0,Y 397.571,Z 534.961,A -85,B 0,C 180,E1 -11339.999,E2 -11339.999} C_VEL
LIN {X 0,Y 397.373,Z 534.986,A -85,B 0,C 180,E1 -11343.041,E2 -11343.041} C_VEL
LIN {X 0,Y 397.348,Z 534.987,A -85,B 0,C 180,E1 -11346.637,E2 -11346.637} C_VEL
LIN {X 0,Y 397.246,Z 535.004,A -85,B 0,C 180,E1 -11349.161,E2 -11349.161} C_VEL
LIN {X 0,Y 397.219,Z 535.005,A -85,B 0,C 180,E1 -11352.258,E2 -11352.258} C_VEL
LIN {X 0,Y 397.168,Z 535.016,A -85,B 0,C 180,E1 -11355.392,E2 -11355.392} C_VEL
LIN {X 0,Y 397.15,Z 535.015,A -85,B 0,C 180,E1 -11358.573,E2 -11358.573} C_VEL
LIN {X 0,Y 397.084,Z 535.022,A -85,B 0,C 180,E1 -11361.819,E2 -11361.819} C_VEL
LIN {X 0,Y 397.171,Z 535.09,A -85,B 0,C 180,E1 -11365.269,E2 -11365.269} C_VEL
LIN {X 0,Y 399.389,Z 546.223,A -85,B 0,C 180,E1 -11368.38,E2 -11368.38} C_VEL
LIN {X 0,Y 399.759,Z 549.288,A -85,B 0,C 180,E1 -11369.199,E2 -11369.199} C_VEL
LIN {X 0,Y 399.636,Z 551.638,A -85,B 0,C 180,E1 -11369.795,E2 -11369.795} C_VEL
LIN {X 0,Y 404.138,Z 573.114,A -85,B 0,C 180,E1 -11370.496,E2 -11370.496} C_VEL
LIN {X 0,Y 402.732,Z 659.387,A -85,B 0,C 180,E1 -11372.157,E2 -11372.157} C_VEL
LIN {X 0,Y 402.257,Z 672.743,A -85,B 0,C 180,E1 -11372.626,E2 -11372.626} C_VEL
LIN {X 0,Y 401.691,Z 684.614,A -85,B 0,C 180,E1 -11373.235,E2 -11373.235} C_VEL
LIN {X 0,Y 400.981,Z 695.409,A -85,B 0,C 180,E1 -11373.966,E2 -11373.966} C_VEL
LIN {X 0,Y 400.211,Z 706.275,A -85,B 0,C 180,E1 -11374.908,E2 -11374.908} C_VEL
LIN {X 0,Y 399.28,Z 717.315,A -85,B 0,C 180,E1 -11376.104,E2 -11376.104} C_VEL
LIN {X 0,Y 398.471,Z 726.723,A -85,B 0,C 180,E1 -11377.374,E2 -11377.374} C_VEL
LIN {X 0,Y 397.722,Z 734.985,A -85,B 0,C 180,E1 -11378.751,E2 -11378.751} C_VEL
LIN {X 0,Y 396.99,Z 743.067,A -85,B 0,C 180,E1 -11380.429,E2 -11380.429} C_VEL
LIN {X 0,Y 396.518,Z 748.665,A -85,B 0,C 180,E1 -11381.893,E2 -11381.893} C_VEL
LIN {X 0,Y 396.238,Z 753.091,A -85,B 0,C 180,E1 -11383.35,E2 -11383.35} C_VEL
LIN {X 0,Y 395.972,Z 756.451,A -85,B 0,C 180,E1 -11384.772,E2 -11384.772} C_VEL
LIN {X 0,Y 395.708,Z 759.691,A -85,B 0,C 180,E1 -11386.733,E2 -11386.733} C_VEL
LIN {X 0,Y 395.578,Z 761.118,A -85,B 0,C 180,E1 -11388.26,E2 -11388.26} C_VEL
LIN {X 0,Y 395.545,Z 761.601,A -85,B 0,C 180,E1 -11390.237,E2 -11390.237} C_VEL
LIN {X 0,Y 395.567,Z 761.123,A -85,B 0,C 180,E1 -11391.552,E2 -11391.552} C_VEL
LIN {X 0,Y 395.654,Z 759.702,A -85,B 0,C 180,E1 -11393.066,E2 -11393.066} C_VEL
LIN {X 0,Y 395.9,Z 757.07,A -85,B 0,C 180,E1 -11394.744,E2 -11394.744} C_VEL
LIN {X 0,Y 396.133,Z 752.624,A -85,B 0,C 180,E1 -11396.636,E2 -11396.636} C_VEL
LIN {X 0,Y 396.52,Z 747.338,A -85,B 0,C 180,E1 -11398.293,E2 -11398.293} C_VEL
LIN {X 0,Y 397.007,Z 740.64,A -85,B 0,C 180,E1 -11399.934,E2 -11399.934} C_VEL
LIN {X 0,Y 397.66,Z 732.512,A -85,B 0,C 180,E1 -11401.5,E2 -11401.5} C_VEL
LIN {X 0,Y 398.447,Z 722.871,A -85,B 0,C 180,E1 -11402.989,E2 -11402.989} C_VEL
LIN {X 0,Y 399.19,Z 713.15,A -85,B 0,C 180,E1 -11404.196,E2 -11404.196} C_VEL
LIN {X 0,Y 400.014,Z 702.294,A -85,B 0,C 180,E1 -11405.276,E2 -11405.276} C_VEL
LIN {X 0,Y 400.739,Z 690.407,A -85,B 0,C 180,E1 -11406.213,E2 -11406.213} C_VEL
LIN {X 0,Y 401.465,Z 678.113,A -85,B 0,C 180,E1 -11406.942,E2 -11406.942} C_VEL
LIN {X 0,Y 402.003,Z 664.89,A -85,B 0,C 180,E1 -11407.498,E2 -11407.498} C_VEL
LIN {X 0,Y 402.312,Z 652.573,A -85,B 0,C 180,E1 -11407.826,E2 -11407.826} C_VEL
LIN {X 0,Y 403.447,Z 572.918,A -85,B 0,C 180,E1 -11409.312,E2 -11409.312} C_VEL
LIN {X 0,Y 399.1,Z 550.919,A -85,B 0,C 180,E1 -11409.952,E2 -11409.952} C_VEL
LIN {X 0,Y 399.299,Z 546.666,A -85,B 0,C 180,E1 -11410.999,E2 -11410.999} C_VEL
LIN {X 0,Y 397.2,Z 535.01,A -85,B 0,C 180,E1 -11414.084,E2 -11414.084} C_VEL
LIN {X 0,Y 397.165,Z 535.011,A -85,B 0,C 180,E1 -11415.227,E2 -11415.227} C_VEL
LIN {X 0,Y 396.509,Z 535.094,A -85,B 0,C 180,E1 -11416.073,E2 -11416.073} C_VEL
LIN {X 0,Y 393.68,Z 535.445,A -85,B 0,C 180,E1 -11417.449,E2 -11417.449} C_VEL
LIN {X 0,Y 391.28,Z 535.745,A -85,B 0,C 180,E1 -11418.56,E2 -11418.56} C_VEL
LIN {X 0,Y 390.247,Z 535.871,A -85,B 0,C 180,E1 -11419.42,E2 -11419.42} C_VEL
LIN {X 0,Y 390.162,Z 535.88,A -85,B 0,C 180,E1 -11419.71,E2 -11419.71} C_VEL
LIN {X 0,Y 390.297,Z 535.87,A -85,B 0,C 180,E1 -11422.76,E2 -11422.76} C_VEL
LIN {X 0,Y 390.222,Z 535.88,A -85,B 0,C 180,E1 -11424.835,E2 -11424.835} C_VEL
LIN {X 0,Y 390.418,Z 535.849,A -85,B 0,C 180,E1 -11427.938,E2 -11427.938} C_VEL
LIN {X 0,Y 390.547,Z 535.832,A -85,B 0,C 180,E1 -11430.001,E2 -11430.001} C_VEL
LIN {X 0,Y 390.312,Z 535.867,A -85,B 0,C 180,E1 -11433.098,E2 -11433.098} C_VEL
LIN {X 0,Y 390.322,Z 535.861,A -85,B 0,C 180,E1 -11436.203,E2 -11436.203} C_VEL
LIN {X 0,Y 390.204,Z 535.879,A -85,B 0,C 180,E1 -11439.33,E2 -11439.33} C_VEL
LIN {X 0,Y 390.193,Z 535.879,A -85,B 0,C 180,E1 -11443.44,E2 -11443.44} C_VEL
LIN {X 0,Y 390.148,Z 535.887,A -85,B 0,C 180,E1 -11447.309,E2 -11447.309} C_VEL
LIN {X 0,Y 390.087,Z 535.891,A -85,B 0,C 180,E1 -11450.472,E2 -11450.472} C_VEL
LIN {X 0,Y 390.09,Z 535.894,A -85,B 0,C 180,E1 -11453.352,E2 -11453.352} C_VEL
LIN {X 0,Y 390.114,Z 535.889,A -85,B 0,C 180,E1 -11456.77,E2 -11456.77} C_VEL
LIN {X 0,Y 390.04,Z 535.896,A -85,B 0,C 180,E1 -11460.301,E2 -11460.301} C_VEL
LIN {X 0,Y 390.07,Z 535.892,A -85,B 0,C 180,E1 -11464.026,E2 -11464.026} C_VEL
LIN {X 0,Y 390.045,Z 535.899,A -85,B 0,C 180,E1 -11467.552,E2 -11467.552} C_VEL
LIN {X 0,Y 390.059,Z 535.895,A -85,B 0,C 180,E1 -11470.823,E2 -11470.823} C_VEL
LIN {X 0,Y 390.06,Z 535.895,A -85,B 0,C 180,E1 -11473.888,E2 -11473.888} C_VEL
LIN {X 0,Y 390.06,Z 535.894,A -85,B 0,C 180,E1 -11476.791,E2 -11476.791} C_VEL
LIN {X 0,Y 390.06,Z 535.899,A -85,B 0,C 180,E1 -11479.562,E2 -11479.562} C_VEL
LIN {X 0,Y 390.047,Z 535.895,A -85,B 0,C 180,E1 -11482.45,E2 -11482.45} C_VEL
LIN {X 0,Y 390.072,Z 535.894,A -85,B 0,C 180,E1 -11485.977,E2 -11485.977} C_VEL
LIN {X 0,Y 390.051,Z 535.897,A -85,B 0,C 180,E1 -11489.87,E2 -11489.87} C_VEL
LIN {X 0,Y 390.118,Z 535.889,A -85,B 0,C 180,E1 -11493.233,E2 -11493.233} C_VEL
LIN {X 0,Y 390.082,Z 535.891,A -85,B 0,C 180,E1 -11496.762,E2 -11496.762} C_VEL
LIN {X 0,Y 390.112,Z 535.89,A -85,B 0,C 180,E1 -11499.984,E2 -11499.984} C_VEL
LIN {X 0,Y 390.144,Z 535.885,A -85,B 0,C 180,E1 -11503.249,E2 -11503.249} C_VEL
LIN {X 0,Y 390.201,Z 535.876,A -85,B 0,C 180,E1 -11506.562,E2 -11506.562} C_VEL
LIN {X 0,Y 390.211,Z 535.874,A -85,B 0,C 180,E1 -11510.672,E2 -11510.672} C_VEL
LIN {X 0,Y 390.331,Z 535.866,A -85,B 0,C 180,E1 -11513.799,E2 -11513.799} C_VEL
LIN {X 0,Y 390.425,Z 535.853,A -85,B 0,C 180,E1 -11517.937,E2 -11517.937} C_VEL
LIN {X 0,Y 390.555,Z 535.837,A -85,B 0,C 180,E1 -11520.001,E2 -11520.001} C_VEL
LIN {X 0,Y 390.317,Z 535.862,A -85,B 0,C 180,E1 -11523.097,E2 -11523.097} C_VEL
LIN {X 0,Y 390.338,Z 535.862,A -85,B 0,C 180,E1 -11526.202,E2 -11526.202} C_VEL
LIN {X 0,Y 390.323,Z 535.863,A -85,B 0,C 180,E1 -11528.282,E2 -11528.282} C_VEL
LIN {X 0,Y 390.178,Z 535.88,A -85,B 0,C 180,E1 -11532.483,E2 -11532.483} C_VEL
LIN {X 0,Y 390.147,Z 535.886,A -85,B 0,C 180,E1 -11535.677,E2 -11535.677} C_VEL
LIN {X 0,Y 390.113,Z 535.887,A -85,B 0,C 180,E1 -11538.922,E2 -11538.922} C_VEL
LIN {X 0,Y 390.046,Z 535.9,A -85,B 0,C 180,E1 -11542.234,E2 -11542.234} C_VEL
LIN {X 0,Y 390.127,Z 535.888,A -85,B 0,C 180,E1 -11545.743,E2 -11545.743} C_VEL
LIN {X 0,Y 390.066,Z 535.892,A -85,B 0,C 180,E1 -11549.109,E2 -11549.109} C_VEL
LIN {X 0,Y 390.051,Z 535.896,A -85,B 0,C 180,E1 -11552.721,E2 -11552.721} C_VEL
LIN {X 0,Y 390.064,Z 535.896,A -85,B 0,C 180,E1 -11555.825,E2 -11555.825} C_VEL
LIN {X 0,Y 390.074,Z 535.891,A -85,B 0,C 180,E1 -11559.217,E2 -11559.217} C_VEL
LIN {X 0,Y 390.047,Z 535.901,A -85,B 0,C 180,E1 -11562.373,E2 -11562.373} C_VEL
LIN {X 0,Y 390.052,Z 535.894,A -85,B 0,C 180,E1 -11565.354,E2 -11565.354} C_VEL
LIN {X 0,Y 390.039,Z 535.901,A -85,B 0,C 180,E1 -11568.186,E2 -11568.186} C_VEL
LIN {X 0,Y 390.1,Z 535.89,A -85,B 0,C 180,E1 -11570.907,E2 -11570.907} C_VEL
LIN {X 0,Y 390.092,Z 535.892,A -85,B 0,C 180,E1 -11574.792,E2 -11574.792} C_VEL
LIN {X 0,Y 390.031,Z 535.904,A -85,B 0,C 180,E1 -11578.495,E2 -11578.495} C_VEL
LIN {X 0,Y 390.154,Z 535.968,A -85,B 0,C 180,E1 -11581.531,E2 -11581.531} C_VEL
LIN {X 0,Y 392.724,Z 548.552,A -85,B 0,C 180,E1 -11584.563,E2 -11584.563} C_VEL
LIN {X 0,Y 393.476,Z 553.641,A -85,B 0,C 180,E1 -11585.743,E2 -11585.743} C_VEL
LIN {X 0,Y 392.376,Z 567.12,A -85,B 0,C 180,E1 -11588.654,E2 -11588.654} C_VEL
LIN {X 0,Y 392.011,Z 572.12,A -85,B 0,C 180,E1 -11589.724,E2 -11589.724} C_VEL
LIN {X 0,Y 396.516,Z 601.207,A -85,B 0,C 180,E1 -11590.523,E2 -11590.523} C_VEL
LIN {X 0,Y 395.317,Z 680.152,A -85,B 0,C 180,E1 -11592.039,E2 -11592.039} C_VEL
LIN {X 0,Y 394.745,Z 693.279,A -85,B 0,C 180,E1 -11592.481,E2 -11592.481} C_VEL
LIN {X 0,Y 394.049,Z 705.416,A -85,B 0,C 180,E1 -11593.084,E2 -11593.084} C_VEL
LIN {X 0,Y 393.276,Z 717.723,A -85,B 0,C 180,E1 -11593.918,E2 -11593.918} C_VEL
LIN {X 0,Y 392.348,Z 729.354,A -85,B 0,C 180,E1 -11594.944,E2 -11594.944} C_VEL
LIN {X 0,Y 391.572,Z 739.712,A -85,B 0,C 180,E1 -11596.093,E2 -11596.093} C_VEL
LIN {X 0,Y 390.874,Z 748.416,A -85,B 0,C 180,E1 -11597.274,E2 -11597.274} C_VEL
LIN {X 0,Y 390.019,Z 757.689,A -85,B 0,C 180,E1 -11598.829,E2 -11598.829} C_VEL
LIN {X 0,Y 389.479,Z 765.144,A -85,B 0,C 180,E1 -11600.39,E2 -11600.39} C_VEL
LIN {X 0,Y 389.033,Z 771.986,A -85,B 0,C 180,E1 -11602.212,E2 -11602.212} C_VEL
LIN {X 0,Y 388.801,Z 776.608,A -85,B 0,C 180,E1 -11603.822,E2 -11603.822} C_VEL
LIN {X 0,Y 388.751,Z 778.859,A -85,B 0,C 180,E1 -11604.812,E2 -11604.812} C_VEL
LIN {X 0,Y 388.704,Z 780.794,A -85,B 0,C 180,E1 -11605.851,E2 -11605.851} C_VEL
LIN {X 0,Y 388.638,Z 782.287,A -85,B 0,C 180,E1 -11606.889,E2 -11606.889} C_VEL
LIN {X 0,Y 388.663,Z 783.329,A -85,B 0,C 180,E1 -11607.926,E2 -11607.926} C_VEL
LIN {X 0,Y 388.704,Z 783.977,A -85,B 0,C 180,E1 -11608.963,E2 -11608.963} C_VEL
LIN {X 0,Y 388.708,Z 784.23,A -85,B 0,C 180,E1 -11609.999,E2 -11609.999} C_VEL
LIN {X 0,Y 388.703,Z 784.067,A -85,B 0,C 180,E1 -11611.035,E2 -11611.035} C_VEL
LIN {X 0,Y 388.661,Z 783.473,A -85,B 0,C 180,E1 -11612.071,E2 -11612.071} C_VEL
LIN {X 0,Y 388.703,Z 781.098,A -85,B 0,C 180,E1 -11614.146,E2 -11614.146} C_VEL
LIN {X 0,Y 388.733,Z 778.055,A -85,B 0,C 180,E1 -11615.76,E2 -11615.76} C_VEL
LIN {X 0,Y 388.938,Z 774.201,A -85,B 0,C 180,E1 -11617.265,E2 -11617.265} C_VEL
LIN {X 0,Y 389.359,Z 768.109,A -85,B 0,C 180,E1 -11619.086,E2 -11619.086} C_VEL
LIN {X 0,Y 389.862,Z 761.425,A -85,B 0,C 180,E1 -11620.646,E2 -11620.646} C_VEL
LIN {X 0,Y 390.64,Z 753.135,A -85,B 0,C 180,E1 -11622.202,E2 -11622.202} C_VEL
LIN {X 0,Y 391.429,Z 744.673,A -85,B 0,C 180,E1 -11623.496,E2 -11623.496} C_VEL
LIN {X 0,Y 392.29,Z 734.492,A -85,B 0,C 180,E1 -11624.763,E2 -11624.763} C_VEL
LIN {X 0,Y 393.298,Z 722.539,A -85,B 0,C 180,E1 -11625.945,E2 -11625.945} C_VEL
LIN {X 0,Y 394.236,Z 710.915,A -85,B 0,C 180,E1 -11626.838,E2 -11626.838} C_VEL
LIN {X 0,Y 395.094,Z 697.612,A -85,B 0,C 180,E1 -11627.6,E2 -11627.6} C_VEL
LIN {X 0,Y 395.769,Z 685.073,A -85,B 0,C 180,E1 -11628.103,E2 -11628.103} C_VEL
LIN {X 0,Y 396.201,Z 670.622,A -85,B 0,C 180,E1 -11628.451,E2 -11628.451} C_VEL
LIN {X 0,Y 397.121,Z 599.969,A -85,B 0,C 180,E1 -11629.821,E2 -11629.821} C_VEL
LIN {X 0,Y 393.622,Z 578.413,A -85,B 0,C 180,E1 -11630.464,E2 -11630.464} C_VEL
LIN {X 0,Y 392.314,Z 571.347,A -85,B 0,C 180,E1 -11630.691,E2 -11630.691} C_VEL
LIN {X 0,Y 393.733,Z 555.171,A -85,B 0,C 180,E1 -11634.237,E2 -11634.237} C_VEL
LIN {X 0,Y 393.12,Z 550.244,A -85,B 0,C 180,E1 -11635.406,E2 -11635.406} C_VEL
LIN {X 0,Y 390.822,Z 539.033,A -85,B 0,C 180,E1 -11638.218,E2 -11638.218} C_VEL
LIN {X 0,Y 390.102,Z 535.896,A -85,B 0,C 180,E1 -11639.04,E2 -11639.04} C_VEL
LIN {X 0,Y 390.039,Z 535.898,A -85,B 0,C 180,E1 -11642.72,E2 -11642.72} C_VEL
LIN {X 0,Y 390.053,Z 535.901,A -85,B 0,C 180,E1 -11645.824,E2 -11645.824} C_VEL
LIN {X 0,Y 390.07,Z 535.901,A -85,B 0,C 180,E1 -11649.218,E2 -11649.218} C_VEL
LIN {X 0,Y 390.076,Z 535.896,A -85,B 0,C 180,E1 -11652.379,E2 -11652.379} C_VEL
LIN {X 0,Y 390.049,Z 535.9,A -85,B 0,C 180,E1 -11656.112,E2 -11656.112} C_VEL
LIN {X 0,Y 390.068,Z 535.895,A -85,B 0,C 180,E1 -11659.561,E2 -11659.561} C_VEL
LIN {X 0,Y 390.04,Z 535.895,A -85,B 0,C 180,E1 -11662.447,E2 -11662.447} C_VEL
LIN {X 0,Y 390.059,Z 535.894,A -85,B 0,C 180,E1 -11666.044,E2 -11666.044} C_VEL
LIN {X 0,Y 390.043,Z 535.899,A -85,B 0,C 180,E1 -11669.866,E2 -11669.866} C_VEL
LIN {X 0,Y 390.104,Z 535.887,A -85,B 0,C 180,E1 -11673.231,E2 -11673.231} C_VEL
LIN {X 0,Y 390.096,Z 535.885,A -85,B 0,C 180,E1 -11676.749,E2 -11676.749} C_VEL
LIN {X 0,Y 390.093,Z 535.885,A -85,B 0,C 180,E1 -11679.982,E2 -11679.982} C_VEL
LIN {X 0,Y 390.127,Z 535.889,A -85,B 0,C 180,E1 -11683.247,E2 -11683.247} C_VEL
LIN {X 0,Y 390.183,Z 535.88,A -85,B 0,C 180,E1 -11686.561,E2 -11686.561} C_VEL
LIN {X 0,Y 390.168,Z 535.886,A -85,B 0,C 180,E1 -11689.622,E2 -11689.622} C_VEL
LIN {X 0,Y 390.307,Z 535.862,A -85,B 0,C 180,E1 -11692.758,E2 -11692.758} C_VEL
LIN {X 0,Y 390.218,Z 535.876,A -85,B 0,C 180,E1 -11694.833,E2 -11694.833} C_VEL
LIN {X 0,Y 390.409,Z 535.85,A -85,B 0,C 180,E1 -11697.936,E2 -11697.936} C_VEL
LIN {X 0,Y 390.54,Z 535.837,A -85,B 0,C 180,E1 -11699.999,E2 -11699.999} C_VEL
LIN {X 0,Y 390.307,Z 535.866,A -85,B 0,C 180,E1 -11703.096,E2 -11703.096} C_VEL
LIN {X 0,Y 390.304,Z 535.864,A -85,B 0,C 180,E1 -11706.633,E2 -11706.633} C_VEL
LIN {X 0,Y 390.198,Z 535.881,A -85,B 0,C 180,E1 -11709.328,E2 -11709.328} C_VEL
LIN {X 0,Y 390.167,Z 535.884,A -85,B 0,C 180,E1 -11712.483,E2 -11712.483} C_VEL
LIN {X 0,Y 390.128,Z 535.892,A -85,B 0,C 180,E1 -11715.677,E2 -11715.677} C_VEL
LIN {X 0,Y 390.093,Z 535.895,A -85,B 0,C 180,E1 -11718.922,E2 -11718.922} C_VEL
LIN {X 0,Y 390.027,Z 535.903,A -85,B 0,C 180,E1 -11722.234,E2 -11722.234} C_VEL
LIN {X 0,Y 390.101,Z 535.914,A -85,B 0,C 180,E1 -11724.905,E2 -11724.905} C_VEL
LIN {X 0,Y 392.164,Z 545.916,A -85,B 0,C 180,E1 -11727.771,E2 -11727.771} C_VEL
LIN {X 0,Y 392.881,Z 549.911,A -85,B 0,C 180,E1 -11728.88,E2 -11728.88} C_VEL
LIN {X 0,Y 392.785,Z 551.923,A -85,B 0,C 180,E1 -11729.401,E2 -11729.401} C_VEL
LIN {X 0,Y 397.491,Z 573.828,A -85,B 0,C 180,E1 -11730.135,E2 -11730.135} C_VEL
LIN {X 0,Y 396.262,Z 649.925,A -85,B 0,C 180,E1 -11731.603,E2 -11731.603} C_VEL
LIN {X 0,Y 395.902,Z 663.815,A -85,B 0,C 180,E1 -11731.942,E2 -11731.942} C_VEL
LIN {X 0,Y 395.384,Z 676.294,A -85,B 0,C 180,E1 -11732.451,E2 -11732.451} C_VEL
LIN {X 0,Y 394.64,Z 688.96,A -85,B 0,C 180,E1 -11733.178,E2 -11733.178} C_VEL
LIN {X 0,Y 393.885,Z 700.304,A -85,B 0,C 180,E1 -11734.042,E2 -11734.042} C_VEL
LIN {X 0,Y 392.986,Z 710.879,A -85,B 0,C 180,E1 -11735.065,E2 -11735.065} C_VEL
LIN {X 0,Y 392.119,Z 720.834,A -85,B 0,C 180,E1 -11736.26,E2 -11736.26} C_VEL
LIN {X 0,Y 391.258,Z 730.167,A -85,B 0,C 180,E1 -11737.641,E2 -11737.641} C_VEL
LIN {X 0,Y 390.51,Z 737.852,A -85,B 0,C 180,E1 -11739.042,E2 -11739.042} C_VEL
LIN {X 0,Y 389.767,Z 745.434,A -85,B 0,C 180,E1 -11740.775,E2 -11740.775} C_VEL
LIN {X 0,Y 389.372,Z 750.605,A -85,B 0,C 180,E1 -11742.269,E2 -11742.269} C_VEL
LIN {X 0,Y 389.071,Z 754.632,A -85,B 0,C 180,E1 -11743.738,E2 -11743.738} C_VEL
LIN {X 0,Y 388.818,Z 757.667,A -85,B 0,C 180,E1 -11745.178,E2 -11745.178} C_VEL
LIN {X 0,Y 388.646,Z 759.831,A -85,B 0,C 180,E1 -11746.596,E2 -11746.596} C_VEL
LIN {X 0,Y 388.524,Z 761.162,A -85,B 0,C 180,E1 -11747.99,E2 -11747.99} C_VEL
LIN {X 0,Y 388.447,Z 761.792,A -85,B 0,C 180,E1 -11749.453,E2 -11749.453} C_VEL
LIN {X 0,Y 388.443,Z 761.562,A -85,B 0,C 180,E1 -11751.076,E2 -11751.076} C_VEL
LIN {X 0,Y 388.544,Z 760.303,A -85,B 0,C 180,E1 -11752.737,E2 -11752.737} C_VEL
LIN {X 0,Y 388.811,Z 757.521,A -85,B 0,C 180,E1 -11754.663,E2 -11754.663} C_VEL
LIN {X 0,Y 388.98,Z 754.179,A -85,B 0,C 180,E1 -11756.212,E2 -11756.212} C_VEL
LIN {X 0,Y 389.356,Z 748.885,A -85,B 0,C 180,E1 -11758.033,E2 -11758.033} C_VEL
LIN {X 0,Y 389.826,Z 742.584,A -85,B 0,C 180,E1 -11759.684,E2 -11759.684} C_VEL
LIN {X 0,Y 390.46,Z 735.534,A -85,B 0,C 180,E1 -11761.163,E2 -11761.163} C_VEL
LIN {X 0,Y 391.042,Z 728.167,A -85,B 0,C 180,E1 -11762.435,E2 -11762.435} C_VEL
LIN {X 0,Y 391.905,Z 718.277,A -85,B 0,C 180,E1 -11763.831,E2 -11763.831} C_VEL
LIN {X 0,Y 392.743,Z 707.973,A -85,B 0,C 180,E1 -11764.993,E2 -11764.993} C_VEL
LIN {X 0,Y 393.567,Z 696.44,A -85,B 0,C 180,E1 -11766.032,E2 -11766.032} C_VEL
LIN {X 0,Y 394.271,Z 684.911,A -85,B 0,C 180,E1 -11766.844,E2 -11766.844} C_VEL
LIN {X 0,Y 394.898,Z 671.932,A -85,B 0,C 180,E1 -11767.514,E2 -11767.514} C_VEL
LIN {X 0,Y 395.369,Z 658.631,A -85,B 0,C 180,E1 -11767.977,E2 -11767.977} C_VEL
LIN {X 0,Y 396.635,Z 573.604,A -85,B 0,C 180,E1 -11769.619,E2 -11769.619} C_VEL
LIN {X 0,Y 392.231,Z 551.043,A -85,B 0,C 180,E1 -11770.303,E2 -11770.303} C_VEL
LIN {X 0,Y 392.285,Z 547.538,A -85,B 0,C 180,E1 -11771.189,E2 -11771.189} C_VEL
LIN {X 0,Y 390.166,Z 535.887,A -85,B 0,C 180,E1 -11774.326,E2 -11774.326} C_VEL
LIN {X 0,Y 390.161,Z 535.883,A -85,B 0,C 180,E1 -11777.518,E2 -11777.518} C_VEL
LIN {X 0,Y 390.162,Z 535.88,A -85,B 0,C 180,E1 -11779.71,E2 -11779.71} C_VEL
LIN {X 0,Y 389.51,Z 535.967,A -85,B 0,C 180,E1 -11780.573,E2 -11780.573} C_VEL
LIN {X 0,Y 386.727,Z 536.309,A -85,B 0,C 180,E1 -11781.977,E2 -11781.977} C_VEL
LIN {X 0,Y 384.354,Z 536.608,A -85,B 0,C 180,E1 -11783.112,E2 -11783.112} C_VEL
LIN {X 0,Y 383.311,Z 536.734,A -85,B 0,C 180,E1 -11783.988,E2 -11783.988} C_VEL
LIN {X 0,Y 383.214,Z 536.747,A -85,B 0,C 180,E1 -11784.284,E2 -11784.284} C_VEL
LIN {X 0,Y 383.385,Z 536.725,A -85,B 0,C 180,E1 -11787.9,E2 -11787.9} C_VEL
LIN {X 0,Y 383.517,Z 536.708,A -85,B 0,C 180,E1 -11790.001,E2 -11790.001} C_VEL
LIN {X 0,Y 383.248,Z 536.746,A -85,B 0,C 180,E1 -11793.155,E2 -11793.155} C_VEL
LIN {X 0,Y 383.278,Z 536.739,A -85,B 0,C 180,E1 -11796.318,E2 -11796.318} C_VEL
LIN {X 0,Y 383.15,Z 536.756,A -85,B 0,C 180,E1 -11799.504,E2 -11799.504} C_VEL
LIN {X 0,Y 383.124,Z 536.759,A -85,B 0,C 180,E1 -11803.538,E2 -11803.538} C_VEL
LIN {X 0,Y 383.094,Z 536.764,A -85,B 0,C 180,E1 -11807.456,E2 -11807.456} C_VEL
LIN {X 0,Y 383.028,Z 536.771,A -85,B 0,C 180,E1 -11810.648,E2 -11810.648} C_VEL
LIN {X 0,Y 383.034,Z 536.769,A -85,B 0,C 180,E1 -11813.809,E2 -11813.809} C_VEL
LIN {X 0,Y 383.08,Z 536.763,A -85,B 0,C 180,E1 -11816.125,E2 -11816.125} C_VEL
LIN {X 0,Y 382.993,Z 536.776,A -85,B 0,C 180,E1 -11819.701,E2 -11819.701} C_VEL
LIN {X 0,Y 383.005,Z 536.778,A -85,B 0,C 180,E1 -11823.402,E2 -11823.402} C_VEL
LIN {X 0,Y 383.034,Z 536.769,A -85,B 0,C 180,E1 -11826.166,E2 -11826.166} C_VEL
LIN {X 0,Y 383.011,Z 536.772,A -85,B 0,C 180,E1 -11829.96,E2 -11829.96} C_VEL
LIN {X 0,Y 383.008,Z 536.773,A -85,B 0,C 180,E1 -11832.78,E2 -11832.78} C_VEL
LIN {X 0,Y 383.001,Z 536.775,A -85,B 0,C 180,E1 -11835.791,E2 -11835.791} C_VEL
LIN {X 0,Y 382.991,Z 536.775,A -85,B 0,C 180,E1 -11838.797,E2 -11838.797} C_VEL
LIN {X 0,Y 383.003,Z 536.773,A -85,B 0,C 180,E1 -11842.098,E2 -11842.098} C_VEL
LIN {X 0,Y 383.022,Z 536.775,A -85,B 0,C 180,E1 -11845.333,E2 -11845.333} C_VEL
LIN {X 0,Y 382.987,Z 536.777,A -85,B 0,C 180,E1 -11849.083,E2 -11849.083} C_VEL
LIN {X 0,Y 383.062,Z 536.765,A -85,B 0,C 180,E1 -11852.699,E2 -11852.699} C_VEL
LIN {X 0,Y 383.056,Z 536.767,A -85,B 0,C 180,E1 -11855.041,E2 -11855.041} C_VEL
LIN {X 0,Y 383.001,Z 536.773,A -85,B 0,C 180,E1 -11858.47,E2 -11858.47} C_VEL
LIN {X 0,Y 383.059,Z 536.77,A -85,B 0,C 180,E1 -11861.827,E2 -11861.827} C_VEL
LIN {X 0,Y 383.116,Z 536.76,A -85,B 0,C 180,E1 -11865.119,E2 -11865.119} C_VEL
LIN {X 0,Y 383.103,Z 536.761,A -85,B 0,C 180,E1 -11868.359,E2 -11868.359} C_VEL
LIN {X 0,Y 383.27,Z 536.743,A -85,B 0,C 180,E1 -11871.977,E2 -11871.977} C_VEL
LIN {X 0,Y 383.204,Z 536.747,A -85,B 0,C 180,E1 -11874.739,E2 -11874.739} C_VEL
LIN {X 0,Y 383.392,Z 536.73,A -85,B 0,C 180,E1 -11877.899,E2 -11877.899} C_VEL
LIN {X 0,Y 383.525,Z 536.712,A -85,B 0,C 180,E1 -11880.001,E2 -11880.001} C_VEL
LIN {X 0,Y 383.253,Z 536.742,A -85,B 0,C 180,E1 -11883.154,E2 -11883.154} C_VEL
LIN {X 0,Y 383.295,Z 536.738,A -85,B 0,C 180,E1 -11886.317,E2 -11886.317} C_VEL
LIN {X 0,Y 383.268,Z 536.741,A -85,B 0,C 180,E1 -11888.436,E2 -11888.436} C_VEL
LIN {X 0,Y 383.144,Z 536.755,A -85,B 0,C 180,E1 -11892.716,E2 -11892.716} C_VEL
LIN {X 0,Y 383.089,Z 536.769,A -85,B 0,C 180,E1 -11895.974,E2 -11895.974} C_VEL
LIN {X 0,Y 383.068,Z 536.765,A -85,B 0,C 180,E1 -11899.284,E2 -11899.284} C_VEL
LIN {X 0,Y 382.999,Z 536.774,A -85,B 0,C 180,E1 -11902.666,E2 -11902.666} C_VEL
LIN {X 0,Y 383.088,Z 536.769,A -85,B 0,C 180,E1 -11906.123,E2 -11906.123} C_VEL
LIN {X 0,Y 383,Z 536.775,A -85,B 0,C 180,E1 -11909.7,E2 -11909.7} C_VEL
LIN {X 0,Y 383.011,Z 536.772,A -85,B 0,C 180,E1 -11913.4,E2 -11913.4} C_VEL
LIN {X 0,Y 383.04,Z 536.775,A -85,B 0,C 180,E1 -11916.164,E2 -11916.164} C_VEL
LIN {X 0,Y 383.015,Z 536.775,A -85,B 0,C 180,E1 -11919.958,E2 -11919.958} C_VEL
LIN {X 0,Y 383.013,Z 536.773,A -85,B 0,C 180,E1 -11922.778,E2 -11922.778} C_VEL
LIN {X 0,Y 383.005,Z 536.774,A -85,B 0,C 180,E1 -11925.789,E2 -11925.789} C_VEL
LIN {X 0,Y 382.996,Z 536.775,A -85,B 0,C 180,E1 -11928.795,E2 -11928.795} C_VEL
LIN {X 0,Y 383.009,Z 536.776,A -85,B 0,C 180,E1 -11932.095,E2 -11932.095} C_VEL
LIN {X 0,Y 383.025,Z 536.77,A -85,B 0,C 180,E1 -11935.331,E2 -11935.331} C_VEL
LIN {X 0,Y 382.99,Z 536.778,A -85,B 0,C 180,E1 -11939.081,E2 -11939.081} C_VEL
LIN {X 0,Y 383.089,Z 536.844,A -85,B 0,C 180,E1 -11941.248,E2 -11941.248} C_VEL
LIN {X 0,Y 385.699,Z 549.484,A -85,B 0,C 180,E1 -11944.356,E2 -11944.356} C_VEL
LIN {X 0,Y 386.415,Z 553.978,A -85,B 0,C 180,E1 -11945.421,E2 -11945.421} C_VEL
LIN {X 0,Y 386.013,Z 560.867,A -85,B 0,C 180,E1 -11946.954,E2 -11946.954} C_VEL
LIN {X 0,Y 385.132,Z 571.864,A -85,B 0,C 180,E1 -11949.363,E2 -11949.363} C_VEL
LIN {X 0,Y 389.739,Z 602.009,A -85,B 0,C 180,E1 -11950.218,E2 -11950.218} C_VEL
LIN {X 0,Y 388.491,Z 680.056,A -85,B 0,C 180,E1 -11951.747,E2 -11951.747} C_VEL
LIN {X 0,Y 387.888,Z 693.898,A -85,B 0,C 180,E1 -11952.229,E2 -11952.229} C_VEL
LIN {X 0,Y 387.168,Z 705.825,A -85,B 0,C 180,E1 -11952.843,E2 -11952.843} C_VEL
LIN {X 0,Y 386.411,Z 717.153,A -85,B 0,C 180,E1 -11953.624,E2 -11953.624} C_VEL
LIN {X 0,Y 385.453,Z 728.855,A -85,B 0,C 180,E1 -11954.669,E2 -11954.669} C_VEL
LIN {X 0,Y 384.613,Z 739.714,A -85,B 0,C 180,E1 -11955.892,E2 -11955.892} C_VEL
LIN {X 0,Y 383.917,Z 748.013,A -85,B 0,C 180,E1 -11957.04,E2 -11957.04} C_VEL
LIN {X 0,Y 383.147,Z 755.948,A -85,B 0,C 180,E1 -11958.358,E2 -11958.358} C_VEL
LIN {X 0,Y 382.524,Z 763.689,A -85,B 0,C 180,E1 -11959.947,E2 -11959.947} C_VEL
LIN {X 0,Y 382.073,Z 769.902,A -85,B 0,C 180,E1 -11961.536,E2 -11961.536} C_VEL
LIN {X 0,Y 381.804,Z 774.825,A -85,B 0,C 180,E1 -11963.127,E2 -11963.127} C_VEL
LIN {X 0,Y 381.654,Z 778.601,A -85,B 0,C 180,E1 -11964.716,E2 -11964.716} C_VEL
LIN {X 0,Y 381.63,Z 780.546,A -85,B 0,C 180,E1 -11965.774,E2 -11965.774} C_VEL
LIN {X 0,Y 381.55,Z 782.054,A -85,B 0,C 180,E1 -11966.831,E2 -11966.831} C_VEL
LIN {X 0,Y 381.562,Z 783.105,A -85,B 0,C 180,E1 -11967.887,E2 -11967.887} C_VEL
LIN {X 0,Y 381.618,Z 783.761,A -85,B 0,C 180,E1 -11968.943,E2 -11968.943} C_VEL
LIN {X 0,Y 381.639,Z 784.021,A -85,B 0,C 180,E1 -11969.998,E2 -11969.998} C_VEL
LIN {X 0,Y 381.603,Z 783.87,A -85,B 0,C 180,E1 -11971.054,E2 -11971.054} C_VEL
LIN {X 0,Y 381.56,Z 783.283,A -85,B 0,C 180,E1 -11972.11,E2 -11972.11} C_VEL
LIN {X 0,Y 381.628,Z 780.919,A -85,B 0,C 180,E1 -11974.223,E2 -11974.223} C_VEL
LIN {X 0,Y 381.673,Z 777.382,A -85,B 0,C 180,E1 -11976.095,E2 -11976.095} C_VEL
LIN {X 0,Y 381.978,Z 772.466,A -85,B 0,C 180,E1 -11977.93,E2 -11977.93} C_VEL
LIN {X 0,Y 382.477,Z 765.93,A -85,B 0,C 180,E1 -11979.784,E2 -11979.784} C_VEL
LIN {X 0,Y 383.066,Z 758.777,A -85,B 0,C 180,E1 -11981.373,E2 -11981.373} C_VEL
LIN {X 0,Y 384.009,Z 749.865,A -85,B 0,C 180,E1 -11982.954,E2 -11982.954} C_VEL
LIN {X 0,Y 384.848,Z 740.471,A -85,B 0,C 180,E1 -11984.308,E2 -11984.308} C_VEL
LIN {X 0,Y 385.784,Z 730.697,A -85,B 0,C 180,E1 -11985.45,E2 -11985.45} C_VEL
LIN {X 0,Y 386.726,Z 719.552,A -85,B 0,C 180,E1 -11986.495,E2 -11986.495} C_VEL
LIN {X 0,Y 387.74,Z 707.101,A -85,B 0,C 180,E1 -11987.4,E2 -11987.4} C_VEL
LIN {X 0,Y 388.521,Z 694.525,A -85,B 0,C 180,E1 -11988.078,E2 -11988.078} C_VEL
LIN {X 0,Y 389.166,Z 681.353,A -85,B 0,C 180,E1 -11988.558,E2 -11988.558} C_VEL
LIN {X 0,Y 389.617,Z 662.178,A -85,B 0,C 180,E1 -11988.967,E2 -11988.967} C_VEL
LIN {X 0,Y 390.526,Z 600.825,A -85,B 0,C 180,E1 -11990.179,E2 -11990.179} C_VEL
LIN {X 0,Y 386.67,Z 577.164,A -85,B 0,C 180,E1 -11990.912,E2 -11990.912} C_VEL
LIN {X 0,Y 385.48,Z 571.085,A -85,B 0,C 180,E1 -11991.128,E2 -11991.128} C_VEL
LIN {X 0,Y 386.88,Z 555.87,A -85,B 0,C 180,E1 -11994.53,E2 -11994.53} C_VEL
LIN {X 0,Y 384.974,Z 545.388,A -85,B 0,C 180,E1 -11997.153,E2 -11997.153} C_VEL
LIN {X 0,Y 383.037,Z 536.778,A -85,B 0,C 180,E1 -11999.467,E2 -11999.467} C_VEL
LIN {X 0,Y 383,Z 536.778,A -85,B 0,C 180,E1 -12003.399,E2 -12003.399} C_VEL
LIN {X 0,Y 383.03,Z 536.775,A -85,B 0,C 180,E1 -12006.163,E2 -12006.163} C_VEL
LIN {X 0,Y 383.015,Z 536.778,A -85,B 0,C 180,E1 -12009.955,E2 -12009.955} C_VEL
LIN {X 0,Y 383.027,Z 536.775,A -85,B 0,C 180,E1 -12012.781,E2 -12012.781} C_VEL
LIN {X 0,Y 382.992,Z 536.782,A -85,B 0,C 180,E1 -12015.788,E2 -12015.788} C_VEL
LIN {X 0,Y 383.008,Z 536.776,A -85,B 0,C 180,E1 -12018.79,E2 -12018.79} C_VEL
LIN {X 0,Y 382.996,Z 536.773,A -85,B 0,C 180,E1 -12022.094,E2 -12022.094} C_VEL
LIN {X 0,Y 383.01,Z 536.774,A -85,B 0,C 180,E1 -12025.331,E2 -12025.331} C_VEL
LIN {X 0,Y 382.978,Z 536.776,A -85,B 0,C 180,E1 -12029.08,E2 -12029.08} C_VEL
LIN {X 0,Y 383.047,Z 536.765,A -85,B 0,C 180,E1 -12032.697,E2 -12032.697} C_VEL
LIN {X 0,Y 383.024,Z 536.766,A -85,B 0,C 180,E1 -12036.192,E2 -12036.192} C_VEL
LIN {X 0,Y 383.045,Z 536.766,A -85,B 0,C 180,E1 -12039.597,E2 -12039.597} C_VEL
LIN {X 0,Y 383.094,Z 536.765,A -85,B 0,C 180,E1 -12042.93,E2 -12042.93} C_VEL
LIN {X 0,Y 383.115,Z 536.761,A -85,B 0,C 180,E1 -12046.463,E2 -12046.463} C_VEL
LIN {X 0,Y 383.13,Z 536.761,A -85,B 0,C 180,E1 -12049.429,E2 -12049.429} C_VEL
LIN {X 0,Y 383.262,Z 536.739,A -85,B 0,C 180,E1 -12052.625,E2 -12052.625} C_VEL
LIN {X 0,Y 383.19,Z 536.751,A -85,B 0,C 180,E1 -12054.738,E2 -12054.738} C_VEL
LIN {X 0,Y 383.377,Z 536.727,A -85,B 0,C 180,E1 -12057.898,E2 -12057.898} C_VEL
LIN {X 0,Y 383.51,Z 536.713,A -85,B 0,C 180,E1 -12059.999,E2 -12059.999} C_VEL
LIN {X 0,Y 383.243,Z 536.747,A -85,B 0,C 180,E1 -12063.153,E2 -12063.153} C_VEL
LIN {X 0,Y 383.264,Z 536.741,A -85,B 0,C 180,E1 -12066.626,E2 -12066.626} C_VEL
LIN {X 0,Y 383.248,Z 536.745,A -85,B 0,C 180,E1 -12068.435,E2 -12068.435} C_VEL
LIN {X 0,Y 383.097,Z 536.765,A -85,B 0,C 180,E1 -12071.642,E2 -12071.642} C_VEL
LIN {X 0,Y 383.1,Z 536.767,A -85,B 0,C 180,E1 -12074.882,E2 -12074.882} C_VEL
LIN {X 0,Y 383.05,Z 536.772,A -85,B 0,C 180,E1 -12078.174,E2 -12078.174} C_VEL
LIN {X 0,Y 382.98,Z 536.778,A -85,B 0,C 180,E1 -12081.531,E2 -12081.531} C_VEL
LIN {X 0,Y 383.018,Z 536.777,A -85,B 0,C 180,E1 -12084.528,E2 -12084.528} C_VEL
LIN {X 0,Y 385.31,Z 547.648,A -85,B 0,C 180,E1 -12087.717,E2 -12087.717} C_VEL
LIN {X 0,Y 385.941,Z 552.088,A -85,B 0,C 180,E1 -12088.959,E2 -12088.959} C_VEL
LIN {X 0,Y 390.366,Z 572.03,A -85,B 0,C 180,E1 -12089.676,E2 -12089.676} C_VEL
LIN {X 0,Y 391.039,Z 577.103,A -85,B 0,C 180,E1 -12089.823,E2 -12089.823} C_VEL
LIN {X 0,Y 389.387,Z 659.644,A -85,B 0,C 180,E1 -12091.466,E2 -12091.466} C_VEL
LIN {X 0,Y 388.844,Z 672.921,A -85,B 0,C 180,E1 -12091.943,E2 -12091.943} C_VEL
LIN {X 0,Y 388.25,Z 684.597,A -85,B 0,C 180,E1 -12092.558,E2 -12092.558} C_VEL
LIN {X 0,Y 387.494,Z 695.705,A -85,B 0,C 180,E1 -12093.33,E2 -12093.33} C_VEL
LIN {X 0,Y 386.598,Z 706.597,A -85,B 0,C 180,E1 -12094.301,E2 -12094.301} C_VEL
LIN {X 0,Y 385.627,Z 717.241,A -85,B 0,C 180,E1 -12095.49,E2 -12095.49} C_VEL
LIN {X 0,Y 384.614,Z 727.587,A -85,B 0,C 180,E1 -12096.935,E2 -12096.935} C_VEL
LIN {X 0,Y 383.705,Z 736.561,A -85,B 0,C 180,E1 -12098.516,E2 -12098.516} C_VEL
LIN {X 0,Y 382.904,Z 744.413,A -85,B 0,C 180,E1 -12100.255,E2 -12100.255} C_VEL
LIN {X 0,Y 382.335,Z 750.626,A -85,B 0,C 180,E1 -12102.038,E2 -12102.038} C_VEL
LIN {X 0,Y 382.047,Z 754.625,A -85,B 0,C 180,E1 -12103.506,E2 -12103.506} C_VEL
LIN {X 0,Y 381.768,Z 757.744,A -85,B 0,C 180,E1 -12104.988,E2 -12104.988} C_VEL
LIN {X 0,Y 381.492,Z 760.598,A -85,B 0,C 180,E1 -12107.031,E2 -12107.031} C_VEL
LIN {X 0,Y 381.38,Z 761.947,A -85,B 0,C 180,E1 -12109.072,E2 -12109.072} C_VEL
LIN {X 0,Y 381.348,Z 761.705,A -85,B 0,C 180,E1 -12111.203,E2 -12111.203} C_VEL
LIN {X 0,Y 381.441,Z 760.731,A -85,B 0,C 180,E1 -12112.556,E2 -12112.556} C_VEL
LIN {X 0,Y 381.612,Z 758.743,A -85,B 0,C 180,E1 -12114.127,E2 -12114.127} C_VEL
LIN {X 0,Y 381.86,Z 755.296,A -85,B 0,C 180,E1 -12115.914,E2 -12115.914} C_VEL
LIN {X 0,Y 382.202,Z 750.276,A -85,B 0,C 180,E1 -12117.776,E2 -12117.776} C_VEL
LIN {X 0,Y 382.656,Z 744.585,A -85,B 0,C 180,E1 -12119.394,E2 -12119.394} C_VEL
LIN {X 0,Y 383.261,Z 737.836,A -85,B 0,C 180,E1 -12120.928,E2 -12120.928} C_VEL
LIN {X 0,Y 383.986,Z 729.339,A -85,B 0,C 180,E1 -12122.476,E2 -12122.476} C_VEL
LIN {X 0,Y 384.781,Z 720.487,A -85,B 0,C 180,E1 -12123.786,E2 -12123.786} C_VEL
LIN {X 0,Y 385.722,Z 709.673,A -85,B 0,C 180,E1 -12125.082,E2 -12125.082} C_VEL
LIN {X 0,Y 386.564,Z 698.33,A -85,B 0,C 180,E1 -12126.154,E2 -12126.154} C_VEL
LIN {X 0,Y 387.364,Z 686.254,A -85,B 0,C 180,E1 -12127.043,E2 -12127.043} C_VEL
LIN {X 0,Y 388.042,Z 673.636,A -85,B 0,C 180,E1 -12127.735,E2 -12127.735} C_VEL
LIN {X 0,Y 388.504,Z 660.732,A -85,B 0,C 180,E1 -12128.217,E2 -12128.217} C_VEL
LIN {X 0,Y 388.898,Z 639.36,A -85,B 0,C 180,E1 -12128.675,E2 -12128.675} C_VEL
LIN {X 0,Y 389.987,Z 575.573,A -85,B 0,C 180,E1 -12129.903,E2 -12129.903} C_VEL
LIN {X 0,Y 385.375,Z 551.173,A -85,B 0,C 180,E1 -12130.666,E2 -12130.666} C_VEL
LIN {X 0,Y 384.923,Z 546.423,A -85,B 0,C 180,E1 -12131.919,E2 -12131.919} C_VEL
LIN {X 0,Y 383.126,Z 536.764,A -85,B 0,C 180,E1 -12134.576,E2 -12134.576} C_VEL
LIN {X 0,Y 383.122,Z 536.762,A -85,B 0,C 180,E1 -12137.285,E2 -12137.285} C_VEL
LIN {X 0,Y 383.147,Z 536.758,A -85,B 0,C 180,E1 -12140.499,E2 -12140.499} C_VEL
LIN {X 0,Y 383.276,Z 536.738,A -85,B 0,C 180,E1 -12143.685,E2 -12143.685} C_VEL
LIN {X 0,Y 383.214,Z 536.747,A -85,B 0,C 180,E1 -12144.284,E2 -12144.284} C_VEL
LIN {X 0,Y 382.505,Z 536.843,A -85,B 0,C 180,E1 -12145.162,E2 -12145.162} C_VEL
LIN {X 0,Y 379.636,Z 537.209,A -85,B 0,C 180,E1 -12146.589,E2 -12146.589} C_VEL
LIN {X 0,Y 377.275,Z 537.503,A -85,B 0,C 180,E1 -12147.742,E2 -12147.742} C_VEL
LIN {X 0,Y 376.326,Z 537.615,A -85,B 0,C 180,E1 -12148.634,E2 -12148.634} C_VEL
LIN {X 0,Y 376.281,Z 537.617,A -85,B 0,C 180,E1 -12148.936,E2 -12148.936} C_VEL
LIN {X 0,Y 376.486,Z 537.584,A -85,B 0,C 180,E1 -12150.002,E2 -12150.002} C_VEL
LIN {X 0,Y 376.186,Z 537.625,A -85,B 0,C 180,E1 -12153.214,E2 -12153.214} C_VEL
LIN {X 0,Y 376.236,Z 537.617,A -85,B 0,C 180,E1 -12156.437,E2 -12156.437} C_VEL
LIN {X 0,Y 376.118,Z 537.631,A -85,B 0,C 180,E1 -12159.683,E2 -12159.683} C_VEL
LIN {X 0,Y 376.088,Z 537.635,A -85,B 0,C 180,E1 -12163.659,E2 -12163.659} C_VEL
LIN {X 0,Y 376.042,Z 537.641,A -85,B 0,C 180,E1 -12167.608,E2 -12167.608} C_VEL
LIN {X 0,Y 375.978,Z 537.651,A -85,B 0,C 180,E1 -12170.834,E2 -12170.834} C_VEL
LIN {X 0,Y 375.994,Z 537.646,A -85,B 0,C 180,E1 -12174.283,E2 -12174.283} C_VEL
LIN {X 0,Y 376.02,Z 537.644,A -85,B 0,C 180,E1 -12176.654,E2 -12176.654} C_VEL
LIN {X 0,Y 375.966,Z 537.649,A -85,B 0,C 180,E1 -12180.314,E2 -12180.314} C_VEL
LIN {X 0,Y 375.961,Z 537.65,A -85,B 0,C 180,E1 -12184.113,E2 -12184.113} C_VEL
LIN {X 0,Y 375.955,Z 537.652,A -85,B 0,C 180,E1 -12186.743,E2 -12186.743} C_VEL
LIN {X 0,Y 375.991,Z 537.647,A -85,B 0,C 180,E1 -12189.972,E2 -12189.972} C_VEL
LIN {X 0,Y 375.934,Z 537.656,A -85,B 0,C 180,E1 -12193.767,E2 -12193.767} C_VEL
LIN {X 0,Y 375.937,Z 537.654,A -85,B 0,C 180,E1 -12196.812,E2 -12196.812} C_VEL
LIN {X 0,Y 375.966,Z 537.649,A -85,B 0,C 180,E1 -12200.539,E2 -12200.539} C_VEL
LIN {X 0,Y 375.967,Z 537.656,A -85,B 0,C 180,E1 -12203.497,E2 -12203.497} C_VEL
LIN {X 0,Y 375.964,Z 537.652,A -85,B 0,C 180,E1 -12205.89,E2 -12205.89} C_VEL
LIN {X 0,Y 375.969,Z 537.654,A -85,B 0,C 180,E1 -12209.688,E2 -12209.688} C_VEL
LIN {X 0,Y 376.001,Z 537.646,A -85,B 0,C 180,E1 -12212.142,E2 -12212.142} C_VEL
LIN {X 0,Y 376.011,Z 537.643,A -85,B 0,C 180,E1 -12214.54,E2 -12214.54} C_VEL
LIN {X 0,Y 375.965,Z 537.651,A -85,B 0,C 180,E1 -12218.047,E2 -12218.047} C_VEL
LIN {X 0,Y 376.009,Z 537.649,A -85,B 0,C 180,E1 -12221.474,E2 -12221.474} C_VEL
LIN {X 0,Y 376.065,Z 537.637,A -85,B 0,C 180,E1 -12224.833,E2 -12224.833} C_VEL
LIN {X 0,Y 376.056,Z 537.64,A -85,B 0,C 180,E1 -12228.137,E2 -12228.137} C_VEL
LIN {X 0,Y 376.226,Z 537.622,A -85,B 0,C 180,E1 -12231.92,E2 -12231.92} C_VEL
LIN {X 0,Y 376.176,Z 537.623,A -85,B 0,C 180,E1 -12234.641,E2 -12234.641} C_VEL
LIN {X 0,Y 376.358,Z 537.607,A -85,B 0,C 180,E1 -12237.86,E2 -12237.86} C_VEL
LIN {X 0,Y 376.494,Z 537.588,A -85,B 0,C 180,E1 -12240.001,E2 -12240.001} C_VEL
LIN {X 0,Y 376.191,Z 537.622,A -85,B 0,C 180,E1 -12243.213,E2 -12243.213} C_VEL
LIN {X 0,Y 376.254,Z 537.615,A -85,B 0,C 180,E1 -12246.435,E2 -12246.435} C_VEL
LIN {X 0,Y 376.213,Z 537.619,A -85,B 0,C 180,E1 -12248.595,E2 -12248.595} C_VEL
LIN {X 0,Y 376.058,Z 537.644,A -85,B 0,C 180,E1 -12251.864,E2 -12251.864} C_VEL
LIN {X 0,Y 376.067,Z 537.637,A -85,B 0,C 180,E1 -12255.168,E2 -12255.168} C_VEL
LIN {X 0,Y 376.032,Z 537.642,A -85,B 0,C 180,E1 -12258.526,E2 -12258.526} C_VEL
LIN {X 0,Y 375.965,Z 537.655,A -85,B 0,C 180,E1 -12261.955,E2 -12261.955} C_VEL
LIN {X 0,Y 376.013,Z 537.644,A -85,B 0,C 180,E1 -12265.461,E2 -12265.461} C_VEL
LIN {X 0,Y 375.969,Z 537.649,A -85,B 0,C 180,E1 -12269.08,E2 -12269.08} C_VEL
LIN {X 0,Y 375.957,Z 537.651,A -85,B 0,C 180,E1 -12272.828,E2 -12272.828} C_VEL
LIN {X 0,Y 375.965,Z 537.649,A -85,B 0,C 180,E1 -12275.415,E2 -12275.415} C_VEL
LIN {X 0,Y 375.98,Z 537.654,A -85,B 0,C 180,E1 -12278.27,E2 -12278.27} C_VEL
LIN {X 0,Y 375.94,Z 537.653,A -85,B 0,C 180,E1 -12281.6,E2 -12281.6} C_VEL
LIN {X 0,Y 375.934,Z 537.653,A -85,B 0,C 180,E1 -12285.268,E2 -12285.268} C_VEL
LIN {X 0,Y 375.942,Z 537.658,A -85,B 0,C 180,E1 -12288.399,E2 -12288.399} C_VEL
LIN {X 0,Y 375.983,Z 537.648,A -85,B 0,C 180,E1 -12291.729,E2 -12291.729} C_VEL
LIN {X 0,Y 375.987,Z 537.646,A -85,B 0,C 180,E1 -12295.332,E2 -12295.332} C_VEL
LIN {X 0,Y 375.965,Z 537.656,A -85,B 0,C 180,E1 -12298.437,E2 -12298.437} C_VEL
LIN {X 0,Y 376.035,Z 537.741,A -85,B 0,C 180,E1 -12300.961,E2 -12300.961} C_VEL
LIN {X 0,Y 378.665,Z 550.395,A -85,B 0,C 180,E1 -12304.139,E2 -12304.139} C_VEL
LIN {X 0,Y 379.494,Z 556.392,A -85,B 0,C 180,E1 -12305.58,E2 -12305.58} C_VEL
LIN {X 0,Y 378.39,Z 569.329,A -85,B 0,C 180,E1 -12308.479,E2 -12308.479} C_VEL
LIN {X 0,Y 378.214,Z 571.966,A -85,B 0,C 180,E1 -12309.022,E2 -12309.022} C_VEL
LIN {X 0,Y 382.969,Z 602.119,A -85,B 0,C 180,E1 -12309.892,E2 -12309.892} C_VEL
LIN {X 0,Y 381.694,Z 679.778,A -85,B 0,C 180,E1 -12311.445,E2 -12311.445} C_VEL
LIN {X 0,Y 381.084,Z 693.642,A -85,B 0,C 180,E1 -12311.936,E2 -12311.936} C_VEL
LIN {X 0,Y 380.292,Z 706.142,A -85,B 0,C 180,E1 -12312.592,E2 -12312.592} C_VEL
LIN {X 0,Y 379.447,Z 718.123,A -85,B 0,C 180,E1 -12313.453,E2 -12313.453} C_VEL
LIN {X 0,Y 378.463,Z 729.617,A -85,B 0,C 180,E1 -12314.516,E2 -12314.516} C_VEL
LIN {X 0,Y 377.623,Z 740.157,A -85,B 0,C 180,E1 -12315.743,E2 -12315.743} C_VEL
LIN {X 0,Y 376.779,Z 749.305,A -85,B 0,C 180,E1 -12317.064,E2 -12317.064} C_VEL
LIN {X 0,Y 375.897,Z 758.344,A -85,B 0,C 180,E1 -12318.677,E2 -12318.677} C_VEL
LIN {X 0,Y 375.315,Z 765.619,A -85,B 0,C 180,E1 -12320.296,E2 -12320.296} C_VEL
LIN {X 0,Y 374.895,Z 771.407,A -85,B 0,C 180,E1 -12321.916,E2 -12321.916} C_VEL
LIN {X 0,Y 374.595,Z 776.843,A -85,B 0,C 180,E1 -12323.919,E2 -12323.919} C_VEL
LIN {X 0,Y 374.556,Z 780.299,A -85,B 0,C 180,E1 -12325.694,E2 -12325.694} C_VEL
LIN {X 0,Y 374.465,Z 781.82,A -85,B 0,C 180,E1 -12326.771,E2 -12326.771} C_VEL
LIN {X 0,Y 374.462,Z 782.881,A -85,B 0,C 180,E1 -12327.847,E2 -12327.847} C_VEL
LIN {X 0,Y 374.518,Z 783.544,A -85,B 0,C 180,E1 -12328.923,E2 -12328.923} C_VEL
LIN {X 0,Y 374.554,Z 783.812,A -85,B 0,C 180,E1 -12329.998,E2 -12329.998} C_VEL
LIN {X 0,Y 374.503,Z 783.673,A -85,B 0,C 180,E1 -12331.074,E2 -12331.074} C_VEL
LIN {X 0,Y 374.459,Z 783.094,A -85,B 0,C 180,E1 -12332.15,E2 -12332.15} C_VEL
LIN {X 0,Y 374.554,Z 780.746,A -85,B 0,C 180,E1 -12334.303,E2 -12334.303} C_VEL
LIN {X 0,Y 374.569,Z 777.596,A -85,B 0,C 180,E1 -12336.045,E2 -12336.045} C_VEL
LIN {X 0,Y 374.804,Z 773.907,A -85,B 0,C 180,E1 -12337.541,E2 -12337.541} C_VEL
LIN {X 0,Y 375.204,Z 768.83,A -85,B 0,C 180,E1 -12339.16,E2 -12339.16} C_VEL
LIN {X 0,Y 375.743,Z 762.461,A -85,B 0,C 180,E1 -12340.779,E2 -12340.779} C_VEL
LIN {X 0,Y 376.576,Z 754.492,A -85,B 0,C 180,E1 -12342.392,E2 -12342.392} C_VEL
LIN {X 0,Y 377.438,Z 746.383,A -85,B 0,C 180,E1 -12343.732,E2 -12343.732} C_VEL
LIN {X 0,Y 378.343,Z 736.504,A -85,B 0,C 180,E1 -12345.072,E2 -12345.072} C_VEL
LIN {X 0,Y 379.42,Z 725.493,A -85,B 0,C 180,E1 -12346.268,E2 -12346.268} C_VEL
LIN {X 0,Y 380.351,Z 714.73,A -85,B 0,C 180,E1 -12347.194,E2 -12347.194} C_VEL
LIN {X 0,Y 381.372,Z 701.834,A -85,B 0,C 180,E1 -12348.047,E2 -12348.047} C_VEL
LIN {X 0,Y 382.157,Z 689.623,A -85,B 0,C 180,E1 -12348.633,E2 -12348.633} C_VEL
LIN {X 0,Y 382.71,Z 675.909,A -85,B 0,C 180,E1 -12349.057,E2 -12349.057} C_VEL
LIN {X 0,Y 383.967,Z 601.715,A -85,B 0,C 180,E1 -12350.556,E2 -12350.556} C_VEL
LIN {X 0,Y 380.048,Z 577.682,A -85,B 0,C 180,E1 -12351.322,E2 -12351.322} C_VEL
LIN {X 0,Y 378.65,Z 570.808,A -85,B 0,C 180,E1 -12351.587,E2 -12351.587} C_VEL
LIN {X 0,Y 379.909,Z 558.118,A -85,B 0,C 180,E1 -12354.482,E2 -12354.482} C_VEL
LIN {X 0,Y 379.461,Z 553.976,A -85,B 0,C 180,E1 -12355.505,E2 -12355.505} C_VEL
LIN {X 0,Y 377.3,Z 543.278,A -85,B 0,C 180,E1 -12358.295,E2 -12358.295} C_VEL
LIN {X 0,Y 375.974,Z 537.66,A -85,B 0,C 180,E1 -12359.846,E2 -12359.846} C_VEL
LIN {X 0,Y 375.946,Z 537.654,A -85,B 0,C 180,E1 -12362.827,E2 -12362.827} C_VEL
LIN {X 0,Y 375.954,Z 537.656,A -85,B 0,C 180,E1 -12365.414,E2 -12365.414} C_VEL
LIN {X 0,Y 375.973,Z 537.654,A -85,B 0,C 180,E1 -12368.27,E2 -12368.27} C_VEL
LIN {X 0,Y 375.956,Z 537.661,A -85,B 0,C 180,E1 -12371.604,E2 -12371.604} C_VEL
LIN {X 0,Y 375.922,Z 537.661,A -85,B 0,C 180,E1 -12375.267,E2 -12375.267} C_VEL
LIN {X 0,Y 375.953,Z 537.654,A -85,B 0,C 180,E1 -12378.393,E2 -12378.393} C_VEL
LIN {X 0,Y 375.971,Z 537.651,A -85,B 0,C 180,E1 -12381.727,E2 -12381.727} C_VEL
LIN {X 0,Y 375.972,Z 537.65,A -85,B 0,C 180,E1 -12385.331,E2 -12385.331} C_VEL
LIN {X 0,Y 375.951,Z 537.651,A -85,B 0,C 180,E1 -12388.437,E2 -12388.437} C_VEL
LIN {X 0,Y 375.993,Z 537.644,A -85,B 0,C 180,E1 -12392.141,E2 -12392.141} C_VEL
LIN {X 0,Y 375.997,Z 537.647,A -85,B 0,C 180,E1 -12394.538,E2 -12394.538} C_VEL
LIN {X 0,Y 375.953,Z 537.654,A -85,B 0,C 180,E1 -12398.045,E2 -12398.045} C_VEL
LIN {X 0,Y 376.013,Z 537.645,A -85,B 0,C 180,E1 -12401.473,E2 -12401.473} C_VEL
LIN {X 0,Y 376.049,Z 537.635,A -85,B 0,C 180,E1 -12404.832,E2 -12404.832} C_VEL
LIN {X 0,Y 376.048,Z 537.636,A -85,B 0,C 180,E1 -12408.136,E2 -12408.136} C_VEL
LIN {X 0,Y 376.246,Z 537.613,A -85,B 0,C 180,E1 -12411.876,E2 -12411.876} C_VEL
LIN {X 0,Y 376.162,Z 537.626,A -85,B 0,C 180,E1 -12414.639,E2 -12414.639} C_VEL
LIN {X 0,Y 376.343,Z 537.603,A -85,B 0,C 180,E1 -12417.859,E2 -12417.859} C_VEL
LIN {X 0,Y 376.479,Z 537.589,A -85,B 0,C 180,E1 -12419.999,E2 -12419.999} C_VEL
LIN {X 0,Y 376.182,Z 537.627,A -85,B 0,C 180,E1 -12423.212,E2 -12423.212} C_VEL
LIN {X 0,Y 376.229,Z 537.618,A -85,B 0,C 180,E1 -12426.615,E2 -12426.615} C_VEL
LIN {X 0,Y 376.194,Z 537.624,A -85,B 0,C 180,E1 -12428.595,E2 -12428.595} C_VEL
LIN {X 0,Y 376.048,Z 537.643,A -85,B 0,C 180,E1 -12431.863,E2 -12431.863} C_VEL
LIN {X 0,Y 376.047,Z 537.647,A -85,B 0,C 180,E1 -12435.167,E2 -12435.167} C_VEL
LIN {X 0,Y 375.996,Z 537.651,A -85,B 0,C 180,E1 -12438.527,E2 -12438.527} C_VEL
LIN {X 0,Y 375.947,Z 537.655,A -85,B 0,C 180,E1 -12441.955,E2 -12441.955} C_VEL
LIN {X 0,Y 376,Z 537.811,A -85,B 0,C 180,E1 -12444.18,E2 -12444.18} C_VEL
LIN {X 0,Y 378.228,Z 548.363,A -85,B 0,C 180,E1 -12447.349,E2 -12447.349} C_VEL
LIN {X 0,Y 378.984,Z 552.418,A -85,B 0,C 180,E1 -12448.523,E2 -12448.523} C_VEL
LIN {X 0,Y 382.069,Z 564.562,A -85,B 0,C 180,E1 -12448.994,E2 -12448.994} C_VEL
LIN {X 0,Y 384.481,Z 576.669,A -85,B 0,C 180,E1 -12449.408,E2 -12449.408} C_VEL
LIN {X 0,Y 382.752,Z 659.604,A -85,B 0,C 180,E1 -12451.092,E2 -12451.092} C_VEL
LIN {X 0,Y 382.18,Z 673.163,A -85,B 0,C 180,E1 -12451.587,E2 -12451.587} C_VEL
LIN {X 0,Y 381.57,Z 684.604,A -85,B 0,C 180,E1 -12452.2,E2 -12452.2} C_VEL
LIN {X 0,Y 380.643,Z 696.916,A -85,B 0,C 180,E1 -12453.08,E2 -12453.08} C_VEL
LIN {X 0,Y 379.602,Z 709.049,A -85,B 0,C 180,E1 -12454.218,E2 -12454.218} C_VEL
LIN {X 0,Y 378.534,Z 719.925,A -85,B 0,C 180,E1 -12455.515,E2 -12455.515} C_VEL
LIN {X 0,Y 377.611,Z 728.883,A -85,B 0,C 180,E1 -12456.844,E2 -12456.844} C_VEL
LIN {X 0,Y 376.705,Z 737.475,A -85,B 0,C 180,E1 -12458.414,E2 -12458.414} C_VEL
LIN {X 0,Y 375.959,Z 744.331,A -85,B 0,C 180,E1 -12459.968,E2 -12459.968} C_VEL
LIN {X 0,Y 375.442,Z 749.816,A -85,B 0,C 180,E1 -12461.519,E2 -12461.519} C_VEL
LIN {X 0,Y 375.077,Z 754.126,A -85,B 0,C 180,E1 -12463.052,E2 -12463.052} C_VEL
LIN {X 0,Y 374.774,Z 757.386,A -85,B 0,C 180,E1 -12464.556,E2 -12464.556} C_VEL
LIN {X 0,Y 374.504,Z 759.737,A -85,B 0,C 180,E1 -12466.027,E2 -12466.027} C_VEL
LIN {X 0,Y 374.377,Z 761.303,A -85,B 0,C 180,E1 -12467.485,E2 -12467.485} C_VEL
LIN {X 0,Y 374.294,Z 762.118,A -85,B 0,C 180,E1 -12468.917,E2 -12468.917} C_VEL
LIN {X 0,Y 374.267,Z 762.191,A -85,B 0,C 180,E1 -12470.344,E2 -12470.344} C_VEL
LIN {X 0,Y 374.295,Z 761.371,A -85,B 0,C 180,E1 -12472.056,E2 -12472.056} C_VEL
LIN {X 0,Y 374.484,Z 759.471,A -85,B 0,C 180,E1 -12473.802,E2 -12473.802} C_VEL
LIN {X 0,Y 374.743,Z 756.02,A -85,B 0,C 180,E1 -12475.765,E2 -12475.765} C_VEL
LIN {X 0,Y 375.046,Z 751.706,A -85,B 0,C 180,E1 -12477.484,E2 -12477.484} C_VEL
LIN {X 0,Y 375.594,Z 745.307,A -85,B 0,C 180,E1 -12479.398,E2 -12479.398} C_VEL
LIN {X 0,Y 376.297,Z 737.584,A -85,B 0,C 180,E1 -12481.191,E2 -12481.191} C_VEL
LIN {X 0,Y 377.12,Z 728.583,A -85,B 0,C 180,E1 -12482.83,E2 -12482.83} C_VEL
LIN {X 0,Y 378.013,Z 718.943,A -85,B 0,C 180,E1 -12484.243,E2 -12484.243} C_VEL
LIN {X 0,Y 378.851,Z 709.497,A -85,B 0,C 180,E1 -12485.365,E2 -12485.365} C_VEL
LIN {X 0,Y 379.679,Z 698.631,A -85,B 0,C 180,E1 -12486.406,E2 -12486.406} C_VEL
LIN {X 0,Y 380.446,Z 687.43,A -85,B 0,C 180,E1 -12487.254,E2 -12487.254} C_VEL
LIN {X 0,Y 381.11,Z 675.661,A -85,B 0,C 180,E1 -12487.933,E2 -12487.933} C_VEL
LIN {X 0,Y 381.664,Z 662.573,A -85,B 0,C 180,E1 -12488.463,E2 -12488.463} C_VEL
LIN {X 0,Y 382.033,Z 646.616,A -85,B 0,C 180,E1 -12488.839,E2 -12488.839} C_VEL
LIN {X 0,Y 383.198,Z 575.753,A -85,B 0,C 180,E1 -12490.238,E2 -12490.238} C_VEL
LIN {X 0,Y 378.451,Z 551.467,A -85,B 0,C 180,E1 -12490.999,E2 -12490.999} C_VEL
LIN {X 0,Y 377.175,Z 543.369,A -85,B 0,C 180,E1 -12493.215,E2 -12493.215} C_VEL
LIN {X 0,Y 376.084,Z 537.64,A -85,B 0,C 180,E1 -12494.835,E2 -12494.835} C_VEL
LIN {X 0,Y 376.042,Z 537.641,A -85,B 0,C 180,E1 -12498.138,E2 -12498.138} C_VEL
LIN {X 0,Y 376.214,Z 537.618,A -85,B 0,C 180,E1 -12501.92,E2 -12501.92} C_VEL
LIN {X 0,Y 376.166,Z 537.628,A -85,B 0,C 180,E1 -12504.641,E2 -12504.641} C_VEL
LIN {X 0,Y 376.351,Z 537.601,A -85,B 0,C 180,E1 -12507.861,E2 -12507.861} C_VEL
LIN {X 0,Y 376.281,Z 537.617,A -85,B 0,C 180,E1 -12508.936,E2 -12508.936} C_VEL
LIN {X 0,Y 375.699,Z 537.683,A -85,B 0,C 180,E1 -12509.83,E2 -12509.83} C_VEL
LIN {X 0,Y 372.844,Z 538.041,A -85,B 0,C 180,E1 -12511.282,E2 -12511.282} C_VEL
LIN {X 0,Y 370.329,Z 538.355,A -85,B 0,C 180,E1 -12512.457,E2 -12512.457} C_VEL
LIN {X 0,Y 369.185,Z 538.497,A -85,B 0,C 180,E1 -12513.366,E2 -12513.366} C_VEL
LIN {X 0,Y 369.061,Z 538.51,A -85,B 0,C 180,E1 -12513.675,E2 -12513.675} C_VEL
LIN {X 0,Y 369.196,Z 538.495,A -85,B 0,C 180,E1 -12516.56,E2 -12516.56} C_VEL
LIN {X 0,Y 369.12,Z 538.506,A -85,B 0,C 180,E1 -12518.763,E2 -12518.763} C_VEL
LIN {X 0,Y 369.004,Z 538.516,A -85,B 0,C 180,E1 -12522.095,E2 -12522.095} C_VEL
LIN {X 0,Y 368.997,Z 538.52,A -85,B 0,C 180,E1 -12525.466,E2 -12525.466} C_VEL
LIN {X 0,Y 368.957,Z 538.526,A -85,B 0,C 180,E1 -12528.896,E2 -12528.896} C_VEL
LIN {X 0,Y 368.932,Z 538.526,A -85,B 0,C 180,E1 -12532.397,E2 -12532.397} C_VEL
LIN {X 0,Y 369.001,Z 538.517,A -85,B 0,C 180,E1 -12535.982,E2 -12535.982} C_VEL
LIN {X 0,Y 368.916,Z 538.529,A -85,B 0,C 180,E1 -12539.692,E2 -12539.692} C_VEL
LIN {X 0,Y 368.898,Z 538.534,A -85,B 0,C 180,E1 -12543.045,E2 -12543.045} C_VEL
LIN {X 0,Y 368.919,Z 538.527,A -85,B 0,C 180,E1 -12546.198,E2 -12546.198} C_VEL
LIN {X 0,Y 368.906,Z 538.531,A -85,B 0,C 180,E1 -12548.954,E2 -12548.954} C_VEL
LIN {X 0,Y 368.884,Z 538.532,A -85,B 0,C 180,E1 -12552.011,E2 -12552.011} C_VEL
LIN {X 0,Y 368.929,Z 538.53,A -85,B 0,C 180,E1 -12555.184,E2 -12555.184} C_VEL
LIN {X 0,Y 368.885,Z 538.531,A -85,B 0,C 180,E1 -12558.179,E2 -12558.179} C_VEL
LIN {X 0,Y 368.912,Z 538.534,A -85,B 0,C 180,E1 -12561.361,E2 -12561.361} C_VEL
LIN {X 0,Y 368.94,Z 538.527,A -85,B 0,C 180,E1 -12565.148,E2 -12565.148} C_VEL
LIN {X 0,Y 368.934,Z 538.527,A -85,B 0,C 180,E1 -12569.048,E2 -12569.048} C_VEL
LIN {X 0,Y 368.985,Z 538.525,A -85,B 0,C 180,E1 -12571.565,E2 -12571.565} C_VEL
LIN {X 0,Y 369.005,Z 538.518,A -85,B 0,C 180,E1 -12574.021,E2 -12574.021} C_VEL
LIN {X 0,Y 368.931,Z 538.532,A -85,B 0,C 180,E1 -12577.605,E2 -12577.605} C_VEL
LIN {X 0,Y 368.961,Z 538.523,A -85,B 0,C 180,E1 -12581.107,E2 -12581.107} C_VEL
LIN {X 0,Y 369.003,Z 538.516,A -85,B 0,C 180,E1 -12584.536,E2 -12584.536} C_VEL
LIN {X 0,Y 369.011,Z 538.52,A -85,B 0,C 180,E1 -12587.908,E2 -12587.908} C_VEL
LIN {X 0,Y 369.173,Z 538.501,A -85,B 0,C 180,E1 -12591.87,E2 -12591.87} C_VEL
LIN {X 0,Y 369.149,Z 538.499,A -85,B 0,C 180,E1 -12594.538,E2 -12594.538} C_VEL
LIN {X 0,Y 369.323,Z 538.483,A -85,B 0,C 180,E1 -12597.819,E2 -12597.819} C_VEL
LIN {X 0,Y 369.464,Z 538.464,A -85,B 0,C 180,E1 -12600.001,E2 -12600.001} C_VEL
LIN {X 0,Y 369.324,Z 538.48,A -85,B 0,C 180,E1 -12602.182,E2 -12602.182} C_VEL
LIN {X 0,Y 369.216,Z 538.491,A -85,B 0,C 180,E1 -12606.559,E2 -12606.559} C_VEL
LIN {X 0,Y 369.145,Z 538.499,A -85,B 0,C 180,E1 -12608.761,E2 -12608.761} C_VEL
LIN {X 0,Y 369.013,Z 538.52,A -85,B 0,C 180,E1 -12612.094,E2 -12612.094} C_VEL
LIN {X 0,Y 369.006,Z 538.518,A -85,B 0,C 180,E1 -12615.465,E2 -12615.465} C_VEL
LIN {X 0,Y 368.975,Z 538.52,A -85,B 0,C 180,E1 -12618.894,E2 -12618.894} C_VEL
LIN {X 0,Y 368.93,Z 538.528,A -85,B 0,C 180,E1 -12622.396,E2 -12622.396} C_VEL
LIN {X 0,Y 369.008,Z 538.521,A -85,B 0,C 180,E1 -12625.98,E2 -12625.98} C_VEL
LIN {X 0,Y 368.923,Z 538.529,A -85,B 0,C 180,E1 -12629.69,E2 -12629.69} C_VEL
LIN {X 0,Y 368.905,Z 538.529,A -85,B 0,C 180,E1 -12633.043,E2 -12633.043} C_VEL
LIN {X 0,Y 368.925,Z 538.533,A -85,B 0,C 180,E1 -12636.197,E2 -12636.197} C_VEL
LIN {X 0,Y 368.908,Z 538.529,A -85,B 0,C 180,E1 -12638.953,E2 -12638.953} C_VEL
LIN {X 0,Y 368.888,Z 538.535,A -85,B 0,C 180,E1 -12642.009,E2 -12642.009} C_VEL
LIN {X 0,Y 368.887,Z 538.531,A -85,B 0,C 180,E1 -12645.175,E2 -12645.175} C_VEL
LIN {X 0,Y 368.891,Z 538.536,A -85,B 0,C 180,E1 -12648.177,E2 -12648.177} C_VEL
LIN {X 0,Y 368.917,Z 538.527,A -85,B 0,C 180,E1 -12651.359,E2 -12651.359} C_VEL
LIN {X 0,Y 368.944,Z 538.524,A -85,B 0,C 180,E1 -12655.146,E2 -12655.146} C_VEL
LIN {X 0,Y 368.936,Z 538.529,A -85,B 0,C 180,E1 -12659.046,E2 -12659.046} C_VEL
LIN {X 0,Y 368.964,Z 538.604,A -85,B 0,C 180,E1 -12660.658,E2 -12660.658} C_VEL
LIN {X 0,Y 371.357,Z 550.016,A -85,B 0,C 180,E1 -12663.592,E2 -12663.592} C_VEL
LIN {X 0,Y 372.553,Z 557.664,A -85,B 0,C 180,E1 -12665.478,E2 -12665.478} C_VEL
LIN {X 0,Y 371.53,Z 569.093,A -85,B 0,C 180,E1 -12668.089,E2 -12668.089} C_VEL
LIN {X 0,Y 371.303,Z 571.503,A -85,B 0,C 180,E1 -12668.634,E2 -12668.634} C_VEL
LIN {X 0,Y 376.226,Z 603.231,A -85,B 0,C 180,E1 -12669.582,E2 -12669.582} C_VEL
LIN {X 0,Y 374.85,Z 680.504,A -85,B 0,C 180,E1 -12671.164,E2 -12671.164} C_VEL
LIN {X 0,Y 374.236,Z 694.061,A -85,B 0,C 180,E1 -12671.664,E2 -12671.664} C_VEL
LIN {X 0,Y 373.413,Z 706.376,A -85,B 0,C 180,E1 -12672.331,E2 -12672.331} C_VEL
LIN {X 0,Y 372.48,Z 719.04,A -85,B 0,C 180,E1 -12673.276,E2 -12673.276} C_VEL
LIN {X 0,Y 371.474,Z 730.332,A -85,B 0,C 180,E1 -12674.358,E2 -12674.358} C_VEL
LIN {X 0,Y 370.653,Z 740.091,A -85,B 0,C 180,E1 -12675.529,E2 -12675.529} C_VEL
LIN {X 0,Y 369.811,Z 748.863,A -85,B 0,C 180,E1 -12676.816,E2 -12676.816} C_VEL
LIN {X 0,Y 368.877,Z 757.944,A -85,B 0,C 180,E1 -12678.459,E2 -12678.459} C_VEL
LIN {X 0,Y 368.277,Z 765.259,A -85,B 0,C 180,E1 -12680.109,E2 -12680.109} C_VEL
LIN {X 0,Y 367.852,Z 771.09,A -85,B 0,C 180,E1 -12681.76,E2 -12681.76} C_VEL
LIN {X 0,Y 367.585,Z 775.665,A -85,B 0,C 180,E1 -12683.411,E2 -12683.411} C_VEL
LIN {X 0,Y 367.477,Z 778.069,A -85,B 0,C 180,E1 -12684.511,E2 -12684.511} C_VEL
LIN {X 0,Y 367.462,Z 780.036,A -85,B 0,C 180,E1 -12685.611,E2 -12685.611} C_VEL
LIN {X 0,Y 367.383,Z 781.574,A -85,B 0,C 180,E1 -12686.708,E2 -12686.708} C_VEL
LIN {X 0,Y 367.363,Z 782.651,A -85,B 0,C 180,E1 -12687.806,E2 -12687.806} C_VEL
LIN {X 0,Y 367.419,Z 783.323,A -85,B 0,C 180,E1 -12688.902,E2 -12688.902} C_VEL
LIN {X 0,Y 367.457,Z 783.601,A -85,B 0,C 180,E1 -12689.998,E2 -12689.998} C_VEL
LIN {X 0,Y 367.403,Z 783.477,A -85,B 0,C 180,E1 -12691.094,E2 -12691.094} C_VEL
LIN {X 0,Y 367.36,Z 782.91,A -85,B 0,C 180,E1 -12692.191,E2 -12692.191} C_VEL
LIN {X 0,Y 367.381,Z 781.944,A -85,B 0,C 180,E1 -12693.288,E2 -12693.288} C_VEL
LIN {X 0,Y 367.46,Z 780.578,A -85,B 0,C 180,E1 -12694.386,E2 -12694.386} C_VEL
LIN {X 0,Y 367.478,Z 777.747,A -85,B 0,C 180,E1 -12696.009,E2 -12696.009} C_VEL
LIN {X 0,Y 367.73,Z 773.771,A -85,B 0,C 180,E1 -12697.687,E2 -12697.687} C_VEL
LIN {X 0,Y 368.167,Z 768.712,A -85,B 0,C 180,E1 -12699.336,E2 -12699.336} C_VEL
LIN {X 0,Y 368.725,Z 762.362,A -85,B 0,C 180,E1 -12700.986,E2 -12700.986} C_VEL
LIN {X 0,Y 369.63,Z 754.424,A -85,B 0,C 180,E1 -12702.628,E2 -12702.628} C_VEL
LIN {X 0,Y 370.524,Z 746.346,A -85,B 0,C 180,E1 -12703.993,E2 -12703.993} C_VEL
LIN {X 0,Y 371.477,Z 736.521,A -85,B 0,C 180,E1 -12705.357,E2 -12705.357} C_VEL
LIN {X 0,Y 372.599,Z 725.604,A -85,B 0,C 180,E1 -12706.574,E2 -12706.574} C_VEL
LIN {X 0,Y 373.747,Z 713.186,A -85,B 0,C 180,E1 -12707.649,E2 -12707.649} C_VEL
LIN {X 0,Y 374.729,Z 701.067,A -85,B 0,C 180,E1 -12708.449,E2 -12708.449} C_VEL
LIN {X 0,Y 375.55,Z 688.549,A -85,B 0,C 180,E1 -12709.044,E2 -12709.044} C_VEL
LIN {X 0,Y 376.104,Z 675.745,A -85,B 0,C 180,E1 -12709.44,E2 -12709.44} C_VEL
LIN {X 0,Y 377.425,Z 602.807,A -85,B 0,C 180,E1 -12710.943,E2 -12710.943} C_VEL
LIN {X 0,Y 373.757,Z 580.026,A -85,B 0,C 180,E1 -12711.688,E2 -12711.688} C_VEL
LIN {X 0,Y 371.829,Z 570.623,A -85,B 0,C 180,E1 -12712.046,E2 -12712.046} C_VEL
LIN {X 0,Y 372.975,Z 560.127,A -85,B 0,C 180,E1 -12714.489,E2 -12714.489} C_VEL
LIN {X 0,Y 372.856,Z 557.205,A -85,B 0,C 180,E1 -12715.208,E2 -12715.208} C_VEL
LIN {X 0,Y 370.822,Z 546.747,A -85,B 0,C 180,E1 -12717.974,E2 -12717.974} C_VEL
LIN {X 0,Y 368.942,Z 538.532,A -85,B 0,C 180,E1 -12720.316,E2 -12720.316} C_VEL
LIN {X 0,Y 368.893,Z 538.536,A -85,B 0,C 180,E1 -12723.536,E2 -12723.536} C_VEL
LIN {X 0,Y 368.899,Z 538.535,A -85,B 0,C 180,E1 -12726.855,E2 -12726.855} C_VEL
LIN {X 0,Y 368.948,Z 538.529,A -85,B 0,C 180,E1 -12730.363,E2 -12730.363} C_VEL
LIN {X 0,Y 368.89,Z 538.541,A -85,B 0,C 180,E1 -12733.616,E2 -12733.616} C_VEL
LIN {X 0,Y 368.897,Z 538.535,A -85,B 0,C 180,E1 -12736.697,E2 -12736.697} C_VEL
LIN {X 0,Y 368.946,Z 538.526,A -85,B 0,C 180,E1 -12739.634,E2 -12739.634} C_VEL
LIN {X 0,Y 368.896,Z 538.53,A -85,B 0,C 180,E1 -12743.142,E2 -12743.142} C_VEL
LIN {X 0,Y 368.888,Z 538.53,A -85,B 0,C 180,E1 -12746.46,E2 -12746.46} C_VEL
LIN {X 0,Y 368.914,Z 538.529,A -85,B 0,C 180,E1 -12750.309,E2 -12750.309} C_VEL
LIN {X 0,Y 368.972,Z 538.521,A -85,B 0,C 180,E1 -12753.534,E2 -12753.534} C_VEL
LIN {X 0,Y 368.957,Z 538.518,A -85,B 0,C 180,E1 -12756.42,E2 -12756.42} C_VEL
LIN {X 0,Y 368.926,Z 538.522,A -85,B 0,C 180,E1 -12759.946,E2 -12759.946} C_VEL
LIN {X 0,Y 368.966,Z 538.522,A -85,B 0,C 180,E1 -12763.398,E2 -12763.398} C_VEL
LIN {X 0,Y 369.049,Z 538.514,A -85,B 0,C 180,E1 -12766.789,E2 -12766.789} C_VEL
LIN {X 0,Y 369.061,Z 538.512,A -85,B 0,C 180,E1 -12770.131,E2 -12770.131} C_VEL
LIN {X 0,Y 369.177,Z 538.493,A -85,B 0,C 180,E1 -12772.342,E2 -12772.342} C_VEL
LIN {X 0,Y 369.135,Z 538.501,A -85,B 0,C 180,E1 -12774.537,E2 -12774.537} C_VEL
LIN {X 0,Y 369.308,Z 538.48,A -85,B 0,C 180,E1 -12777.818,E2 -12777.818} C_VEL
LIN {X 0,Y 369.449,Z 538.465,A -85,B 0,C 180,E1 -12779.999,E2 -12779.999} C_VEL
LIN {X 0,Y 369.308,Z 538.479,A -85,B 0,C 180,E1 -12782.181,E2 -12782.181} C_VEL
LIN {X 0,Y 369.199,Z 538.495,A -85,B 0,C 180,E1 -12786.602,E2 -12786.602} C_VEL
LIN {X 0,Y 369.127,Z 538.505,A -85,B 0,C 180,E1 -12788.761,E2 -12788.761} C_VEL
LIN {X 0,Y 369.002,Z 538.521,A -85,B 0,C 180,E1 -12792.093,E2 -12792.093} C_VEL
LIN {X 0,Y 368.986,Z 538.526,A -85,B 0,C 180,E1 -12795.465,E2 -12795.465} C_VEL
LIN {X 0,Y 368.945,Z 538.529,A -85,B 0,C 180,E1 -12798.894,E2 -12798.894} C_VEL
LIN {X 0,Y 368.918,Z 538.533,A -85,B 0,C 180,E1 -12802.395,E2 -12802.395} C_VEL
LIN {X 0,Y 368.975,Z 538.702,A -85,B 0,C 180,E1 -12803.772,E2 -12803.772} C_VEL
LIN {X 0,Y 371.227,Z 549.253,A -85,B 0,C 180,E1 -12807.023,E2 -12807.023} C_VEL
LIN {X 0,Y 371.864,Z 552.632,A -85,B 0,C 180,E1 -12808.026,E2 -12808.026} C_VEL
LIN {X 0,Y 374.154,Z 559.605,A -85,B 0,C 180,E1 -12808.351,E2 -12808.351} C_VEL
LIN {X 0,Y 377.85,Z 577.07,A -85,B 0,C 180,E1 -12808.991,E2 -12808.991} C_VEL
LIN {X 0,Y 376.135,Z 659.956,A -85,B 0,C 180,E1 -12810.714,E2 -12810.714} C_VEL
LIN {X 0,Y 375.571,Z 672.884,A -85,B 0,C 180,E1 -12811.191,E2 -12811.191} C_VEL
LIN {X 0,Y 374.874,Z 685.017,A -85,B 0,C 180,E1 -12811.847,E2 -12811.847} C_VEL
LIN {X 0,Y 373.938,Z 697.005,A -85,B 0,C 180,E1 -12812.72,E2 -12812.72} C_VEL
LIN {X 0,Y 372.872,Z 708.931,A -85,B 0,C 180,E1 -12813.854,E2 -12813.854} C_VEL
LIN {X 0,Y 371.853,Z 718.854,A -85,B 0,C 180,E1 -12815.035,E2 -12815.035} C_VEL
LIN {X 0,Y 370.945,Z 727.193,A -85,B 0,C 180,E1 -12816.248,E2 -12816.248} C_VEL
LIN {X 0,Y 370.004,Z 735.601,A -85,B 0,C 180,E1 -12817.741,E2 -12817.741} C_VEL
LIN {X 0,Y 369.229,Z 742.508,A -85,B 0,C 180,E1 -12819.247,E2 -12819.247} C_VEL
LIN {X 0,Y 368.505,Z 749.416,A -85,B 0,C 180,E1 -12821.138,E2 -12821.138} C_VEL
LIN {X 0,Y 368.068,Z 753.788,A -85,B 0,C 180,E1 -12822.675,E2 -12822.675} C_VEL
LIN {X 0,Y 367.748,Z 757.217,A -85,B 0,C 180,E1 -12824.223,E2 -12824.223} C_VEL
LIN {X 0,Y 367.461,Z 759.725,A -85,B 0,C 180,E1 -12825.751,E2 -12825.751} C_VEL
LIN {X 0,Y 367.247,Z 761.904,A -85,B 0,C 180,E1 -12827.951,E2 -12827.951} C_VEL
LIN {X 0,Y 367.158,Z 762.456,A -85,B 0,C 180,E1 -12829.965,E2 -12829.965} C_VEL
LIN {X 0,Y 367.185,Z 761.85,A -85,B 0,C 180,E1 -12831.696,E2 -12831.696} C_VEL
LIN {X 0,Y 367.357,Z 759.961,A -85,B 0,C 180,E1 -12833.627,E2 -12833.627} C_VEL
LIN {X 0,Y 367.601,Z 757.294,A -85,B 0,C 180,E1 -12835.294,E2 -12835.294} C_VEL
LIN {X 0,Y 367.884,Z 752.961,A -85,B 0,C 180,E1 -12837.199,E2 -12837.199} C_VEL
LIN {X 0,Y 368.419,Z 746.995,A -85,B 0,C 180,E1 -12839.139,E2 -12839.139} C_VEL
LIN {X 0,Y 369.029,Z 740.557,A -85,B 0,C 180,E1 -12840.76,E2 -12840.76} C_VEL
LIN {X 0,Y 369.698,Z 733.302,A -85,B 0,C 180,E1 -12842.243,E2 -12842.243} C_VEL
LIN {X 0,Y 370.615,Z 723.646,A -85,B 0,C 180,E1 -12843.841,E2 -12843.841} C_VEL
LIN {X 0,Y 371.574,Z 713.238,A -85,B 0,C 180,E1 -12845.212,E2 -12845.212} C_VEL
LIN {X 0,Y 372.562,Z 702.194,A -85,B 0,C 180,E1 -12846.37,E2 -12846.37} C_VEL
LIN {X 0,Y 373.398,Z 690.032,A -85,B 0,C 180,E1 -12847.376,E2 -12847.376} C_VEL
LIN {X 0,Y 374.237,Z 677.2,A -85,B 0,C 180,E1 -12848.159,E2 -12848.159} C_VEL
LIN {X 0,Y 374.816,Z 664.761,A -85,B 0,C 180,E1 -12848.699,E2 -12848.699} C_VEL
LIN {X 0,Y 375.205,Z 651.98,A -85,B 0,C 180,E1 -12849.046,E2 -12849.046} C_VEL
LIN {X 0,Y 376.514,Z 577.279,A -85,B 0,C 180,E1 -12850.547,E2 -12850.547} C_VEL
LIN {X 0,Y 371.953,Z 553.662,A -85,B 0,C 180,E1 -12851.296,E2 -12851.296} C_VEL
LIN {X 0,Y 371.416,Z 551.633,A -85,B 0,C 180,E1 -12851.381,E2 -12851.381} C_VEL
LIN {X 0,Y 369.408,Z 540.384,A -85,B 0,C 180,E1 -12854.555,E2 -12854.555} C_VEL
LIN {X 0,Y 369.022,Z 538.521,A -85,B 0,C 180,E1 -12855.103,E2 -12855.103} C_VEL
LIN {X 0,Y 368.998,Z 538.519,A -85,B 0,C 180,E1 -12857.908,E2 -12857.908} C_VEL
LIN {X 0,Y 369.183,Z 538.494,A -85,B 0,C 180,E1 -12861.847,E2 -12861.847} C_VEL
LIN {X 0,Y 369.139,Z 538.503,A -85,B 0,C 180,E1 -12864.539,E2 -12864.539} C_VEL
LIN {X 0,Y 369.316,Z 538.477,A -85,B 0,C 180,E1 -12867.82,E2 -12867.82} C_VEL
LIN {X 0,Y 369.456,Z 538.46,A -85,B 0,C 180,E1 -12870.002,E2 -12870.002} C_VEL
LIN {X 0,Y 369.316,Z 538.478,A -85,B 0,C 180,E1 -12872.183,E2 -12872.183} C_VEL
LIN {X 0,Y 369.061,Z 538.51,A -85,B 0,C 180,E1 -12873.675,E2 -12873.675} C_VEL
LIN {X 0,Y 368.343,Z 538.603,A -85,B 0,C 180,E1 -12874.587,E2 -12874.587} C_VEL
LIN {X 0,Y 365.579,Z 538.943,A -85,B 0,C 180,E1 -12876.072,E2 -12876.072} C_VEL
LIN {X 0,Y 363.254,Z 539.236,A -85,B 0,C 180,E1 -12877.273,E2 -12877.273} C_VEL
LIN {X 0,Y 362.214,Z 539.363,A -85,B 0,C 180,E1 -12878.2,E2 -12878.2} C_VEL
LIN {X 0,Y 362.103,Z 539.378,A -85,B 0,C 180,E1 -12878.513,E2 -12878.513} C_VEL
LIN {X 0,Y 361.959,Z 539.394,A -85,B 0,C 180,E1 -12882.334,E2 -12882.334} C_VEL
LIN {X 0,Y 361.961,Z 539.396,A -85,B 0,C 180,E1 -12884.622,E2 -12884.622} C_VEL
LIN {X 0,Y 361.955,Z 539.394,A -85,B 0,C 180,E1 -12888.101,E2 -12888.101} C_VEL
LIN {X 0,Y 361.892,Z 539.404,A -85,B 0,C 180,E1 -12891.654,E2 -12891.654} C_VEL
LIN {X 0,Y 361.929,Z 539.403,A -85,B 0,C 180,E1 -12895.292,E2 -12895.292} C_VEL
LIN {X 0,Y 361.909,Z 539.401,A -85,B 0,C 180,E1 -12897.78,E2 -12897.78} C_VEL
LIN {X 0,Y 361.839,Z 539.411,A -85,B 0,C 180,E1 -12901.631,E2 -12901.631} C_VEL
LIN {X 0,Y 361.876,Z 539.41,A -85,B 0,C 180,E1 -12905.346,E2 -12905.346} C_VEL
LIN {X 0,Y 361.872,Z 539.408,A -85,B 0,C 180,E1 -12909.028,E2 -12909.028} C_VEL
LIN {X 0,Y 361.84,Z 539.41,A -85,B 0,C 180,E1 -12912.83,E2 -12912.83} C_VEL
LIN {X 0,Y 361.838,Z 539.41,A -85,B 0,C 180,E1 -12915.945,E2 -12915.945} C_VEL
LIN {X 0,Y 361.839,Z 539.414,A -85,B 0,C 180,E1 -12919.246,E2 -12919.246} C_VEL
LIN {X 0,Y 361.867,Z 539.406,A -85,B 0,C 180,E1 -12922.778,E2 -12922.778} C_VEL
LIN {X 0,Y 361.858,Z 539.41,A -85,B 0,C 180,E1 -12925.721,E2 -12925.721} C_VEL
LIN {X 0,Y 361.879,Z 539.409,A -85,B 0,C 180,E1 -12929.673,E2 -12929.673} C_VEL
LIN {X 0,Y 361.96,Z 539.4,A -85,B 0,C 180,E1 -12933.476,E2 -12933.476} C_VEL
LIN {X 0,Y 361.888,Z 539.405,A -85,B 0,C 180,E1 -12937.145,E2 -12937.145} C_VEL
LIN {X 0,Y 361.893,Z 539.402,A -85,B 0,C 180,E1 -12940.723,E2 -12940.723} C_VEL
LIN {X 0,Y 361.95,Z 539.396,A -85,B 0,C 180,E1 -12944.227,E2 -12944.227} C_VEL
LIN {X 0,Y 362.005,Z 539.388,A -85,B 0,C 180,E1 -12946.529,E2 -12946.529} C_VEL
LIN {X 0,Y 362.038,Z 539.388,A -85,B 0,C 180,E1 -12949.939,E2 -12949.939} C_VEL
LIN {X 0,Y 362.168,Z 539.37,A -85,B 0,C 180,E1 -12953.314,E2 -12953.314} C_VEL
LIN {X 0,Y 362.287,Z 539.36,A -85,B 0,C 180,E1 -12957.777,E2 -12957.777} C_VEL
LIN {X 0,Y 362.434,Z 539.34,A -85,B 0,C 180,E1 -12960.001,E2 -12960.001} C_VEL
LIN {X 0,Y 362.288,Z 539.356,A -85,B 0,C 180,E1 -12962.224,E2 -12962.224} C_VEL
LIN {X 0,Y 362.18,Z 539.367,A -85,B 0,C 180,E1 -12966.687,E2 -12966.687} C_VEL
LIN {X 0,Y 362.082,Z 539.379,A -85,B 0,C 180,E1 -12968.934,E2 -12968.934} C_VEL
LIN {X 0,Y 361.968,Z 539.395,A -85,B 0,C 180,E1 -12972.333,E2 -12972.333} C_VEL
LIN {X 0,Y 361.97,Z 539.393,A -85,B 0,C 180,E1 -12974.621,E2 -12974.621} C_VEL
LIN {X 0,Y 361.966,Z 539.399,A -85,B 0,C 180,E1 -12978.1,E2 -12978.1} C_VEL
LIN {X 0,Y 361.869,Z 539.408,A -85,B 0,C 180,E1 -12981.655,E2 -12981.655} C_VEL
LIN {X 0,Y 361.935,Z 539.397,A -85,B 0,C 180,E1 -12985.29,E2 -12985.29} C_VEL
LIN {X 0,Y 361.917,Z 539.402,A -85,B 0,C 180,E1 -12987.779,E2 -12987.779} C_VEL
LIN {X 0,Y 361.846,Z 539.41,A -85,B 0,C 180,E1 -12991.629,E2 -12991.629} C_VEL
LIN {X 0,Y 361.882,Z 539.404,A -85,B 0,C 180,E1 -12995.344,E2 -12995.344} C_VEL
LIN {X 0,Y 361.875,Z 539.405,A -85,B 0,C 180,E1 -12999.026,E2 -12999.026} C_VEL
LIN {X 0,Y 361.843,Z 539.41,A -85,B 0,C 180,E1 -13002.828,E2 -13002.828} C_VEL
LIN {X 0,Y 361.826,Z 539.413,A -85,B 0,C 180,E1 -13005.946,E2 -13005.946} C_VEL
LIN {X 0,Y 361.844,Z 539.408,A -85,B 0,C 180,E1 -13009.244,E2 -13009.244} C_VEL
LIN {X 0,Y 361.879,Z 539.406,A -85,B 0,C 180,E1 -13012.775,E2 -13012.775} C_VEL
LIN {X 0,Y 361.862,Z 539.407,A -85,B 0,C 180,E1 -13015.719,E2 -13015.719} C_VEL
LIN {X 0,Y 361.888,Z 539.407,A -85,B 0,C 180,E1 -13019.672,E2 -13019.672} C_VEL
LIN {X 0,Y 361.927,Z 539.491,A -85,B 0,C 180,E1 -13020.355,E2 -13020.355} C_VEL
LIN {X 0,Y 364.58,Z 552.174,A -85,B 0,C 180,E1 -13023.679,E2 -13023.679} C_VEL
LIN {X 0,Y 365.576,Z 558.554,A -85,B 0,C 180,E1 -13025.282,E2 -13025.282} C_VEL
LIN {X 0,Y 364.495,Z 570.557,A -85,B 0,C 180,E1 -13028.076,E2 -13028.076} C_VEL
LIN {X 0,Y 364.431,Z 571.497,A -85,B 0,C 180,E1 -13028.268,E2 -13028.268} C_VEL
LIN {X 0,Y 369.466,Z 603.604,A -85,B 0,C 180,E1 -13029.243,E2 -13029.243} C_VEL
